LIN {X 0,Y 368.03,Z 575.323,A -85,B 0,C 180,E1 10655.932,E2 10655.932} C_VEL
LIN {X 0,Y 372.432,Z 552.778,A -85,B 0,C 180,E1 10654.833,E2 10654.833} C_VEL
LIN {X 0,Y 375.58,Z 532.541,A -85,B 0,C 180,E1 10654.081,E2 10654.081} C_VEL
LIN {X 0,Y 378.339,Z 507.8,A -85,B 0,C 180,E1 10653.405,E2 10653.405} C_VEL
LIN {X 0,Y 390.575,Z 315.874,A -85,B 0,C 180,E1 10649.482,E2 10649.482} C_VEL
LIN {X 0,Y 393.17,Z 275.11,A -85,B 0,C 180,E1 10648.652,E2 10648.652} C_VEL
LIN {X 0,Y 384.379,Z 261.212,A -85,B 0,C 180,E1 10645.871,E2 10645.871} C_VEL
LIN {X 0,Y 376.778,Z 250,A -85,B 0,C 180,E1 10643.167,E2 10643.167} C_VEL
LIN {X 0,Y 370.187,Z 240.873,A -85,B 0,C 180,E1 10640.515,E2 10640.515} C_VEL
LIN {X 0,Y 365.396,Z 234.593,A -85,B 0,C 180,E1 10638.341,E2 10638.341} C_VEL
LIN {X 0,Y 362.255,Z 230.576,A -85,B 0,C 180,E1 10636.764,E2 10636.764} C_VEL
LIN {X 0,Y 358.691,Z 226.093,A -85,B 0,C 180,E1 10634.777,E2 10634.777} C_VEL
LIN {X 0,Y 354.481,Z 220.931,A -85,B 0,C 180,E1 10632.047,E2 10632.047} C_VEL
LIN {X 0,Y 349.673,Z 215.334,A -85,B 0,C 180,E1 10628.054,E2 10628.054} C_VEL
LIN {X 0,Y 344.902,Z 210.541,A -85,B 0,C 180,E1 10620.996,E2 10620.996} C_VEL
LIN {X 0,Y 344.302,Z 209.98,A -85,B 0,C 180,E1 10617.836,E2 10617.836} C_VEL
LIN {X 0,Y 344.699,Z 211.471,A -85,B 0,C 180,E1 10614.006,E2 10614.006} C_VEL
LIN {X 0,Y 347.562,Z 215.069,A -85,B 0,C 180,E1 10608.799,E2 10608.799} C_VEL
LIN {X 0,Y 350.867,Z 219.711,A -85,B 0,C 180,E1 10605.308,E2 10605.308} C_VEL
LIN {X 0,Y 351.984,Z 221.296,A -85,B 0,C 180,E1 10604.344,E2 10604.344} C_VEL
LIN {X 0,Y 355.628,Z 226.333,A -85,B 0,C 180,E1 10601.645,E2 10601.645} C_VEL
LIN {X 0,Y 359.331,Z 231.448,A -85,B 0,C 180,E1 10599.348,E2 10599.348} C_VEL
LIN {X 0,Y 363.967,Z 237.983,A -85,B 0,C 180,E1 10596.869,E2 10596.869} C_VEL
LIN {X 0,Y 370.087,Z 246.981,A -85,B 0,C 180,E1 10594.044,E2 10594.044} C_VEL
LIN {X 0,Y 376.169,Z 256.349,A -85,B 0,C 180,E1 10591.589,E2 10591.589} C_VEL
LIN {X 0,Y 382.889,Z 267.209,A -85,B 0,C 180,E1 10589.171,E2 10589.171} C_VEL
LIN {X 0,Y 389.905,Z 279.202,A -85,B 0,C 180,E1 10586.892,E2 10586.892} C_VEL
LIN {X 0,Y 390.523,Z 280.623,A -85,B 0,C 180,E1 10586.69,E2 10586.69} C_VEL
LIN {X 0,Y 377.585,Z 508.657,A -85,B 0,C 180,E1 10582.319,E2 10582.319} C_VEL
LIN {X 0,Y 375.428,Z 530.973,A -85,B 0,C 180,E1 10581.772,E2 10581.772} C_VEL
LIN {X 0,Y 372.339,Z 551.704,A -85,B 0,C 180,E1 10581.048,E2 10581.048} C_VEL
LIN {X 0,Y 368.361,Z 572.767,A -85,B 0,C 180,E1 10580.066,E2 10580.066} C_VEL
LIN {X 0,Y 364.024,Z 591.67,A -85,B 0,C 180,E1 10578.945,E2 10578.945} C_VEL
LIN {X 0,Y 358.708,Z 611.311,A -85,B 0,C 180,E1 10577.497,E2 10577.497} C_VEL
LIN {X 0,Y 353.173,Z 629.571,A -85,B 0,C 180,E1 10575.857,E2 10575.857} C_VEL
LIN {X 0,Y 346.964,Z 647.622,A -85,B 0,C 180,E1 10573.871,E2 10573.871} C_VEL
LIN {X 0,Y 340.274,Z 665.618,A -85,B 0,C 180,E1 10571.471,E2 10571.471} C_VEL
LIN {X 0,Y 333.892,Z 681.773,A -85,B 0,C 180,E1 10568.868,E2 10568.868} C_VEL
LIN {X 0,Y 327.863,Z 696.153,A -85,B 0,C 180,E1 10566.055,E2 10566.055} C_VEL
LIN {X 0,Y 321.867,Z 710.299,A -85,B 0,C 180,E1 10562.718,E2 10562.718} C_VEL
LIN {X 0,Y 316.825,Z 722.338,A -85,B 0,C 180,E1 10559.284,E2 10559.284} C_VEL
LIN {X 0,Y 312.53,Z 732.875,A -85,B 0,C 180,E1 10555.587,E2 10555.587} C_VEL
LIN {X 0,Y 309.109,Z 742.014,A -85,B 0,C 180,E1 10551.638,E2 10551.638} C_VEL
LIN {X 0,Y 306.717,Z 749.426,A -85,B 0,C 180,E1 10547.647,E2 10547.647} C_VEL
LIN {X 0,Y 305.203,Z 755.071,A -85,B 0,C 180,E1 10543.643,E2 10543.643} C_VEL
LIN {X 0,Y 304.379,Z 759.395,A -85,B 0,C 180,E1 10539.453,E2 10539.453} C_VEL
LIN {X 0,Y 304.077,Z 761.943,A -85,B 0,C 180,E1 10535.661,E2 10535.661} C_VEL
LIN {X 0,Y 303.986,Z 763.224,A -85,B 0,C 180,E1 10531.696,E2 10531.696} C_VEL
LIN {X 0,Y 303.989,Z 763.215,A -85,B 0,C 180,E1 10528.115,E2 10528.115} C_VEL
LIN {X 0,Y 304.083,Z 761.893,A -85,B 0,C 180,E1 10524.15,E2 10524.15} C_VEL
LIN {X 0,Y 304.392,Z 759.324,A -85,B 0,C 180,E1 10520.356,E2 10520.356} C_VEL
LIN {X 0,Y 305.236,Z 754.954,A -85,B 0,C 180,E1 10516.165,E2 10516.165} C_VEL
LIN {X 0,Y 306.324,Z 750.737,A -85,B 0,C 180,E1 10513.119,E2 10513.119} C_VEL
LIN {X 0,Y 306.002,Z 748.668,A -85,B 0,C 180,E1 10511.721,E2 10511.721} C_VEL
LIN {X 0,Y 302.102,Z 742.719,A -85,B 0,C 180,E1 10507.942,E2 10507.942} C_VEL
LIN {X 0,Y 302.28,Z 740.45,A -85,B 0,C 180,E1 10506.752,E2 10506.752} C_VEL
LIN {X 0,Y 306.107,Z 730.963,A -85,B 0,C 180,E1 10502.788,E2 10502.788} C_VEL
LIN {X 0,Y 311.162,Z 719.337,A -85,B 0,C 180,E1 10498.847,E2 10498.847} C_VEL
LIN {X 0,Y 316.773,Z 706.845,A -85,B 0,C 180,E1 10495.38,E2 10495.38} C_VEL
LIN {X 0,Y 322.621,Z 693.621,A -85,B 0,C 180,E1 10492.373,E2 10492.373} C_VEL
LIN {X 0,Y 329.225,Z 678.283,A -85,B 0,C 180,E1 10489.466,E2 10489.466} C_VEL
LIN {X 0,Y 335.931,Z 662.054,A -85,B 0,C 180,E1 10486.917,E2 10486.917} C_VEL
LIN {X 0,Y 342.314,Z 645.186,A -85,B 0,C 180,E1 10484.744,E2 10484.744} C_VEL
LIN {X 0,Y 349.073,Z 625.729,A -85,B 0,C 180,E1 10482.674,E2 10482.674} C_VEL
LIN {X 0,Y 355.034,Z 606.549,A -85,B 0,C 180,E1 10481.01,E2 10481.01} C_VEL
LIN {X 0,Y 360.276,Z 586.779,A -85,B 0,C 180,E1 10479.636,E2 10479.636} C_VEL
LIN {X 0,Y 365.159,Z 564.965,A -85,B 0,C 180,E1 10478.43,E2 10478.43} C_VEL
LIN {X 0,Y 369.101,Z 543.179,A -85,B 0,C 180,E1 10477.517,E2 10477.517} C_VEL
LIN {X 0,Y 371.952,Z 521.251,A -85,B 0,C 180,E1 10476.867,E2 10476.867} C_VEL
LIN {X 0,Y 374.108,Z 491.918,A -85,B 0,C 180,E1 10476.246,E2 10476.246} C_VEL
LIN {X 0,Y 386.33,Z 284.515,A -85,B 0,C 180,E1 10472.262,E2 10472.262} C_VEL
LIN {X 0,Y 378.451,Z 270.786,A -85,B 0,C 180,E1 10469.564,E2 10469.564} C_VEL
LIN {X 0,Y 370.714,Z 258.332,A -85,B 0,C 180,E1 10466.555,E2 10466.555} C_VEL
LIN {X 0,Y 364.99,Z 249.636,A -85,B 0,C 180,E1 10464.004,E2 10464.004} C_VEL
LIN {X 0,Y 359.677,Z 241.804,A -85,B 0,C 180,E1 10461.271,E2 10461.271} C_VEL
LIN {X 0,Y 356.149,Z 236.756,A -85,B 0,C 180,E1 10459.176,E2 10459.176} C_VEL
LIN {X 0,Y 352.925,Z 232.202,A -85,B 0,C 180,E1 10456.966,E2 10456.966} C_VEL
LIN {X 0,Y 349.827,Z 227.657,A -85,B 0,C 180,E1 10454.398,E2 10454.398} C_VEL
LIN {X 0,Y 346.535,Z 223.028,A -85,B 0,C 180,E1 10450.81,E2 10450.81} C_VEL
LIN {X 0,Y 344.076,Z 219.991,A -85,B 0,C 180,E1 10446.34,E2 10446.34} C_VEL
LIN {X 0,Y 343.53,Z 218.311,A -85,B 0,C 180,E1 10442.336,E2 10442.336} C_VEL
LIN {X 0,Y 344.064,Z 218.755,A -85,B 0,C 180,E1 10439.168,E2 10439.168} C_VEL
LIN {X 0,Y 348.217,Z 222.986,A -85,B 0,C 180,E1 10432.576,E2 10432.576} C_VEL
LIN {X 0,Y 349.257,Z 224.156,A -85,B 0,C 180,E1 10431.522,E2 10431.522} C_VEL
LIN {X 0,Y 354.086,Z 229.86,A -85,B 0,C 180,E1 10427.608,E2 10427.608} C_VEL
LIN {X 0,Y 358.751,Z 235.756,A -85,B 0,C 180,E1 10424.647,E2 10424.647} C_VEL
LIN {X 0,Y 363.139,Z 241.45,A -85,B 0,C 180,E1 10422.287,E2 10422.287} C_VEL
LIN {X 0,Y 369.123,Z 249.401,A -85,B 0,C 180,E1 10419.507,E2 10419.507} C_VEL
LIN {X 0,Y 376.122,Z 259.55,A -85,B 0,C 180,E1 10416.666,E2 10416.666} C_VEL
LIN {X 0,Y 383.714,Z 271.114,A -85,B 0,C 180,E1 10413.956,E2 10413.956} C_VEL
LIN {X 0,Y 388.89,Z 279.747,A -85,B 0,C 180,E1 10412.261,E2 10412.261} C_VEL
LIN {X 0,Y 375.193,Z 488.195,A -85,B 0,C 180,E1 10408.022,E2 10408.022} C_VEL
LIN {X 0,Y 372.711,Z 518.69,A -85,B 0,C 180,E1 10407.334,E2 10407.334} C_VEL
LIN {X 0,Y 369.596,Z 541.745,A -85,B 0,C 180,E1 10406.622,E2 10406.622} C_VEL
LIN {X 0,Y 365.445,Z 564.474,A -85,B 0,C 180,E1 10405.646,E2 10405.646} C_VEL
LIN {X 0,Y 360.248,Z 587.797,A -85,B 0,C 180,E1 10404.349,E2 10404.349} C_VEL
LIN {X 0,Y 354.809,Z 608.696,A -85,B 0,C 180,E1 10402.89,E2 10402.89} C_VEL
LIN {X 0,Y 348.682,Z 629.121,A -85,B 0,C 180,E1 10401.125,E2 10401.125} C_VEL
LIN {X 0,Y 342.163,Z 648.952,A -85,B 0,C 180,E1 10399.057,E2 10399.057} C_VEL
LIN {X 0,Y 335.831,Z 666.622,A -85,B 0,C 180,E1 10396.837,E2 10396.837} C_VEL
LIN {X 0,Y 328.72,Z 685.312,A -85,B 0,C 180,E1 10394.027,E2 10394.027} C_VEL
LIN {X 0,Y 322.316,Z 701.724,A -85,B 0,C 180,E1 10391.079,E2 10391.079} C_VEL
LIN {X 0,Y 316.265,Z 716.75,A -85,B 0,C 180,E1 10387.829,E2 10387.829} C_VEL
LIN {X 0,Y 310.526,Z 731.331,A -85,B 0,C 180,E1 10384.073,E2 10384.073} C_VEL
LIN {X 0,Y 305.865,Z 743.789,A -85,B 0,C 180,E1 10380.225,E2 10380.225} C_VEL
LIN {X 0,Y 302.198,Z 754.312,A -85,B 0,C 180,E1 10376.282,E2 10376.282} C_VEL
LIN {X 0,Y 299.451,Z 763.498,A -85,B 0,C 180,E1 10372.166,E2 10372.166} C_VEL
LIN {X 0,Y 297.611,Z 770.879,A -85,B 0,C 180,E1 10368.004,E2 10368.004} C_VEL
LIN {X 0,Y 296.523,Z 776.987,A -85,B 0,C 180,E1 10363.652,E2 10363.652} C_VEL
LIN {X 0,Y 296.094,Z 780.812,A -85,B 0,C 180,E1 10359.917,E2 10359.917} C_VEL
LIN {X 0,Y 295.973,Z 783.478,A -85,B 0,C 180,E1 10356.206,E2 10356.206} C_VEL
LIN {X 0,Y 295.966,Z 784.977,A -85,B 0,C 180,E1 10352.13,E2 10352.13} C_VEL
LIN {X 0,Y 295.971,Z 785.074,A -85,B 0,C 180,E1 10348.645,E2 10348.645} C_VEL
LIN {X 0,Y 295.956,Z 784.128,A -85,B 0,C 180,E1 10345.155,E2 10345.155} C_VEL
LIN {X 0,Y 296.038,Z 781.654,A -85,B 0,C 180,E1 10341.062,E2 10341.062} C_VEL
LIN {X 0,Y 296.38,Z 778.076,A -85,B 0,C 180,E1 10337.334,E2 10337.334} C_VEL
LIN {X 0,Y 297.238,Z 772.774,A -85,B 0,C 180,E1 10333.185,E2 10333.185} C_VEL
LIN {X 0,Y 298.868,Z 765.608,A -85,B 0,C 180,E1 10328.969,E2 10328.969} C_VEL
LIN {X 0,Y 301.477,Z 756.611,A -85,B 0,C 180,E1 10324.671,E2 10324.671} C_VEL
LIN {X 0,Y 304.866,Z 746.485,A -85,B 0,C 180,E1 10320.737,E2 10320.737} C_VEL
LIN {X 0,Y 309.498,Z 733.937,A -85,B 0,C 180,E1 10316.689,E2 10316.689} C_VEL
LIN {X 0,Y 314.73,Z 720.655,A -85,B 0,C 180,E1 10313.101,E2 10313.101} C_VEL
LIN {X 0,Y 320.576,Z 705.886,A -85,B 0,C 180,E1 10309.789,E2 10309.789} C_VEL
LIN {X 0,Y 327.099,Z 689.449,A -85,B 0,C 180,E1 10306.677,E2 10306.677} C_VEL
LIN {X 0,Y 333.306,Z 673.234,A -85,B 0,C 180,E1 10304.103,E2 10304.103} C_VEL
LIN {X 0,Y 340.192,Z 654.371,A -85,B 0,C 180,E1 10301.597,E2 10301.597} C_VEL
LIN {X 0,Y 346.634,Z 635.528,A -85,B 0,C 180,E1 10299.504,E2 10299.504} C_VEL
LIN {X 0,Y 352.633,Z 615.965,A -85,B 0,C 180,E1 10297.716,E2 10297.716} C_VEL
LIN {X 0,Y 358.134,Z 596.262,A -85,B 0,C 180,E1 10296.213,E2 10296.213} C_VEL
LIN {X 0,Y 363.003,Z 575.753,A -85,B 0,C 180,E1 10294.954,E2 10294.954} C_VEL
LIN {X 0,Y 367.47,Z 553.785,A -85,B 0,C 180,E1 10293.874,E2 10293.874} C_VEL
LIN {X 0,Y 370.785,Z 533.196,A -85,B 0,C 180,E1 10293.103,E2 10293.103} C_VEL
LIN {X 0,Y 373.66,Z 508.504,A -85,B 0,C 180,E1 10292.422,E2 10292.422} C_VEL
LIN {X 0,Y 386.203,Z 318.554,A -85,B 0,C 180,E1 10288.527,E2 10288.527} C_VEL
LIN {X 0,Y 388.714,Z 279.297,A -85,B 0,C 180,E1 10287.705,E2 10287.705} C_VEL
LIN {X 0,Y 380.162,Z 265.668,A -85,B 0,C 180,E1 10284.858,E2 10284.858} C_VEL
LIN {X 0,Y 371.938,Z 253.409,A -85,B 0,C 180,E1 10281.734,E2 10281.734} C_VEL
LIN {X 0,Y 364.697,Z 243.494,A -85,B 0,C 180,E1 10278.543,E2 10278.543} C_VEL
LIN {X 0,Y 360.39,Z 237.928,A -85,B 0,C 180,E1 10276.355,E2 10276.355} C_VEL
LIN {X 0,Y 357.044,Z 233.634,A -85,B 0,C 180,E1 10274.432,E2 10274.432} C_VEL
LIN {X 0,Y 353.047,Z 228.624,A -85,B 0,C 180,E1 10271.765,E2 10271.765} C_VEL
LIN {X 0,Y 348.527,Z 223.207,A -85,B 0,C 180,E1 10267.915,E2 10267.915} C_VEL
LIN {X 0,Y 343.873,Z 218.424,A -85,B 0,C 180,E1 10260.833,E2 10260.833} C_VEL
LIN {X 0,Y 343.32,Z 217.931,A -85,B 0,C 180,E1 10257.663,E2 10257.663} C_VEL
LIN {X 0,Y 343.825,Z 219.685,A -85,B 0,C 180,E1 10253.655,E2 10253.655} C_VEL
LIN {X 0,Y 346.399,Z 222.9,A -85,B 0,C 180,E1 10249.017,E2 10249.017} C_VEL
LIN {X 0,Y 349.73,Z 227.605,A -85,B 0,C 180,E1 10245.428,E2 10245.428} C_VEL
LIN {X 0,Y 354.082,Z 233.9,A -85,B 0,C 180,E1 10241.988,E2 10241.988} C_VEL
LIN {X 0,Y 357.7,Z 239.039,A -85,B 0,C 180,E1 10239.677,E2 10239.677} C_VEL
LIN {X 0,Y 362.132,Z 245.409,A -85,B 0,C 180,E1 10237.244,E2 10237.244} C_VEL
LIN {X 0,Y 368.105,Z 254.397,A -85,B 0,C 180,E1 10234.413,E2 10234.413} C_VEL
LIN {X 0,Y 374.923,Z 265.093,A -85,B 0,C 180,E1 10231.617,E2 10231.617} C_VEL
LIN {X 0,Y 382.618,Z 278.019,A -85,B 0,C 180,E1 10228.841,E2 10228.841} C_VEL
LIN {X 0,Y 386.222,Z 284.81,A -85,B 0,C 180,E1 10227.633,E2 10227.633} C_VEL
LIN {X 0,Y 372.875,Z 510.263,A -85,B 0,C 180,E1 10223.289,E2 10223.289} C_VEL
LIN {X 0,Y 370.464,Z 533.064,A -85,B 0,C 180,E1 10222.709,E2 10222.709} C_VEL
LIN {X 0,Y 367.326,Z 553.251,A -85,B 0,C 180,E1 10221.99,E2 10221.99} C_VEL
LIN {X 0,Y 363.3,Z 573.556,A -85,B 0,C 180,E1 10221.029,E2 10221.029} C_VEL
LIN {X 0,Y 358.531,Z 593.601,A -85,B 0,C 180,E1 10219.827,E2 10219.827} C_VEL
LIN {X 0,Y 352.879,Z 613.422,A -85,B 0,C 180,E1 10218.328,E2 10218.328} C_VEL
LIN {X 0,Y 346.543,Z 633.073,A -85,B 0,C 180,E1 10216.496,E2 10216.496} C_VEL
LIN {X 0,Y 340.245,Z 650.696,A -85,B 0,C 180,E1 10214.495,E2 10214.495} C_VEL
LIN {X 0,Y 333.634,Z 667.524,A -85,B 0,C 180,E1 10212.166,E2 10212.166} C_VEL
LIN {X 0,Y 326.963,Z 683.557,A -85,B 0,C 180,E1 10209.498,E2 10209.498} C_VEL
LIN {X 0,Y 320.947,Z 697.338,A -85,B 0,C 180,E1 10206.736,E2 10206.736} C_VEL
LIN {X 0,Y 315.012,Z 710.641,A -85,B 0,C 180,E1 10203.523,E2 10203.523} C_VEL
LIN {X 0,Y 309.701,Z 722.665,A -85,B 0,C 180,E1 10200.026,E2 10200.026} C_VEL
LIN {X 0,Y 305.16,Z 733.199,A -85,B 0,C 180,E1 10196.252,E2 10196.252} C_VEL
LIN {X 0,Y 301.52,Z 742.327,A -85,B 0,C 180,E1 10192.211,E2 10192.211} C_VEL
LIN {X 0,Y 298.956,Z 749.731,A -85,B 0,C 180,E1 10188.121,E2 10188.121} C_VEL
LIN {X 0,Y 297.323,Z 755.373,A -85,B 0,C 180,E1 10184.012,E2 10184.012} C_VEL
LIN {X 0,Y 296.427,Z 759.691,A -85,B 0,C 180,E1 10179.709,E2 10179.709} C_VEL
LIN {X 0,Y 296.093,Z 762.237,A -85,B 0,C 180,E1 10175.814,E2 10175.814} C_VEL
LIN {X 0,Y 295.992,Z 763.515,A -85,B 0,C 180,E1 10171.742,E2 10171.742} C_VEL
LIN {X 0,Y 295.994,Z 763.526,A -85,B 0,C 180,E1 10168.258,E2 10168.258} C_VEL
LIN {X 0,Y 296.089,Z 762.292,A -85,B 0,C 180,E1 10164.186,E2 10164.186} C_VEL
LIN {X 0,Y 296.412,Z 759.769,A -85,B 0,C 180,E1 10160.29,E2 10160.29} C_VEL
LIN {X 0,Y 297.359,Z 755.254,A -85,B 0,C 180,E1 10155.791,E2 10155.791} C_VEL
LIN {X 0,Y 299.015,Z 749.588,A -85,B 0,C 180,E1 10151.681,E2 10151.681} C_VEL
LIN {X 0,Y 301.605,Z 742.133,A -85,B 0,C 180,E1 10147.59,E2 10147.59} C_VEL
LIN {X 0,Y 302.28,Z 740.45,A -85,B 0,C 180,E1 10146.752,E2 10146.752} C_VEL
LIN {X 0,Y 302.486,Z 737.71,A -85,B 0,C 180,E1 10145.376,E2 10145.376} C_VEL
LIN {X 0,Y 300.12,Z 730.017,A -85,B 0,C 180,E1 10141.634,E2 10141.634} C_VEL
LIN {X 0,Y 300.759,Z 727.058,A -85,B 0,C 180,E1 10140.501,E2 10140.501} C_VEL
LIN {X 0,Y 306.243,Z 715.364,A -85,B 0,C 180,E1 10136.736,E2 10136.736} C_VEL
LIN {X 0,Y 312.14,Z 702.702,A -85,B 0,C 180,E1 10133.431,E2 10133.431} C_VEL
LIN {X 0,Y 319.23,Z 687.304,A -85,B 0,C 180,E1 10130.118,E2 10130.118} C_VEL
LIN {X 0,Y 326.173,Z 671.688,A -85,B 0,C 180,E1 10127.356,E2 10127.356} C_VEL
LIN {X 0,Y 332.899,Z 655.333,A -85,B 0,C 180,E1 10124.984,E2 10124.984} C_VEL
LIN {X 0,Y 339.889,Z 636.967,A -85,B 0,C 180,E1 10122.783,E2 10122.783} C_VEL
LIN {X 0,Y 346.384,Z 618.198,A -85,B 0,C 180,E1 10120.939,E2 10120.939} C_VEL
LIN {X 0,Y 352.092,Z 599.148,A -85,B 0,C 180,E1 10119.431,E2 10119.431} C_VEL
LIN {X 0,Y 357.576,Z 578.029,A -85,B 0,C 180,E1 10118.084,E2 10118.084} C_VEL
LIN {X 0,Y 361.727,Z 558.766,A -85,B 0,C 180,E1 10117.115,E2 10117.115} C_VEL
LIN {X 0,Y 365.378,Z 537.264,A -85,B 0,C 180,E1 10116.297,E2 10116.297} C_VEL
LIN {X 0,Y 368.092,Z 515.346,A -85,B 0,C 180,E1 10115.693,E2 10115.693} C_VEL
LIN {X 0,Y 375.18,Z 399.549,A -85,B 0,C 180,E1 10113.432,E2 10113.432} C_VEL
LIN {X 0,Y 382.145,Z 288.685,A -85,B 0,C 180,E1 10111.298,E2 10111.298} C_VEL
LIN {X 0,Y 374.329,Z 275.003,A -85,B 0,C 180,E1 10108.476,E2 10108.476} C_VEL
LIN {X 0,Y 366.684,Z 262.542,A -85,B 0,C 180,E1 10105.304,E2 10105.304} C_VEL
LIN {X 0,Y 360.625,Z 253.213,A -85,B 0,C 180,E1 10102.367,E2 10102.367} C_VEL
LIN {X 0,Y 357.213,Z 248.275,A -85,B 0,C 180,E1 10100.48,E2 10100.48} C_VEL
LIN {X 0,Y 354.454,Z 244.161,A -85,B 0,C 180,E1 10098.758,E2 10098.758} C_VEL
LIN {X 0,Y 351.322,Z 239.643,A -85,B 0,C 180,E1 10096.535,E2 10096.535} C_VEL
LIN {X 0,Y 348.335,Z 235.208,A -85,B 0,C 180,E1 10093.952,E2 10093.952} C_VEL
LIN {X 0,Y 345.275,Z 230.594,A -85,B 0,C 180,E1 10090.428,E2 10090.428} C_VEL
LIN {X 0,Y 342.577,Z 226.627,A -85,B 0,C 180,E1 10083.682,E2 10083.682} C_VEL
LIN {X 0,Y 342.76,Z 226.314,A -85,B 0,C 180,E1 10080.502,E2 10080.502} C_VEL
LIN {X 0,Y 344.521,Z 228.504,A -85,B 0,C 180,E1 10076.006,E2 10076.006} C_VEL
LIN {X 0,Y 347.865,Z 231.702,A -85,B 0,C 180,E1 10071.904,E2 10071.904} C_VEL
LIN {X 0,Y 352.641,Z 237.555,A -85,B 0,C 180,E1 10067.889,E2 10067.889} C_VEL
LIN {X 0,Y 357.085,Z 243.288,A -85,B 0,C 180,E1 10064.989,E2 10064.989} C_VEL
LIN {X 0,Y 361.383,Z 248.999,A -85,B 0,C 180,E1 10062.614,E2 10062.614} C_VEL
LIN {X 0,Y 367.013,Z 256.652,A -85,B 0,C 180,E1 10059.924,E2 10059.924} C_VEL
LIN {X 0,Y 373.867,Z 266.827,A -85,B 0,C 180,E1 10057.059,E2 10057.059} C_VEL
LIN {X 0,Y 381.029,Z 277.988,A -85,B 0,C 180,E1 10054.427,E2 10054.427} C_VEL
LIN {X 0,Y 384.609,Z 284.061,A -85,B 0,C 180,E1 10053.207,E2 10053.207} C_VEL
LIN {X 0,Y 370.454,Z 492.545,A -85,B 0,C 180,E1 10048.958,E2 10048.958} C_VEL
LIN {X 0,Y 368.064,Z 519.686,A -85,B 0,C 180,E1 10048.331,E2 10048.331} C_VEL
LIN {X 0,Y 364.839,Z 542.581,A -85,B 0,C 180,E1 10047.618,E2 10047.618} C_VEL
LIN {X 0,Y 360.591,Z 565.067,A -85,B 0,C 180,E1 10046.646,E2 10046.646} C_VEL
LIN {X 0,Y 355.227,Z 588.262,A -85,B 0,C 180,E1 10045.35,E2 10045.35} C_VEL
LIN {X 0,Y 349.525,Z 609.415,A -85,B 0,C 180,E1 10043.865,E2 10043.865} C_VEL
LIN {X 0,Y 343.279,Z 629.417,A -85,B 0,C 180,E1 10042.121,E2 10042.121} C_VEL
LIN {X 0,Y 336.52,Z 649.173,A -85,B 0,C 180,E1 10040.044,E2 10040.044} C_VEL
LIN {X 0,Y 330.017,Z 666.624,A -85,B 0,C 180,E1 10037.832,E2 10037.832} C_VEL
LIN {X 0,Y 322.785,Z 684.85,A -85,B 0,C 180,E1 10035.07,E2 10035.07} C_VEL
LIN {X 0,Y 316.095,Z 701.184,A -85,B 0,C 180,E1 10032.111,E2 10032.111} C_VEL
LIN {X 0,Y 309.671,Z 716.386,A -85,B 0,C 180,E1 10028.782,E2 10028.782} C_VEL
LIN {X 0,Y 303.597,Z 730.986,A -85,B 0,C 180,E1 10024.962,E2 10024.962} C_VEL
LIN {X 0,Y 298.86,Z 742.852,A -85,B 0,C 180,E1 10021.235,E2 10021.235} C_VEL
LIN {X 0,Y 294.759,Z 753.905,A -85,B 0,C 180,E1 10017.035,E2 10017.035} C_VEL
LIN {X 0,Y 291.776,Z 763.182,A -85,B 0,C 180,E1 10012.781,E2 10012.781} C_VEL
LIN {X 0,Y 289.773,Z 770.568,A -85,B 0,C 180,E1 10008.508,E2 10008.508} C_VEL
LIN {X 0,Y 288.586,Z 776.685,A -85,B 0,C 180,E1 10004.035,E2 10004.035} C_VEL
LIN {X 0,Y 288.112,Z 780.514,A -85,B 0,C 180,E1 10000.194,E2 10000.194} C_VEL
LIN {X 0,Y 287.98,Z 783.184,A -85,B 0,C 180,E1 9996.379,E2 9996.379} C_VEL
LIN {X 0,Y 287.972,Z 784.686,A -85,B 0,C 180,E1 9992.189,E2 9992.189} C_VEL
LIN {X 0,Y 287.976,Z 784.783,A -85,B 0,C 180,E1 9988.607,E2 9988.607} C_VEL
LIN {X 0,Y 287.96,Z 783.835,A -85,B 0,C 180,E1 9985.02,E2 9985.02} C_VEL
LIN {X 0,Y 288.052,Z 781.355,A -85,B 0,C 180,E1 9980.812,E2 9980.812} C_VEL
LIN {X 0,Y 288.433,Z 777.719,A -85,B 0,C 180,E1 9976.928,E2 9976.928} C_VEL
LIN {X 0,Y 289.435,Z 772.15,A -85,B 0,C 180,E1 9972.51,E2 9972.51} C_VEL
LIN {X 0,Y 291.204,Z 765.021,A -85,B 0,C 180,E1 9968.234,E2 9968.234} C_VEL
LIN {X 0,Y 294.101,Z 755.802,A -85,B 0,C 180,E1 9963.772,E2 9963.772} C_VEL
LIN {X 0,Y 297.565,Z 746.177,A -85,B 0,C 180,E1 9959.957,E2 9959.957} C_VEL
LIN {X 0,Y 302.512,Z 733.586,A -85,B 0,C 180,E1 9955.815,E2 9955.815} C_VEL
LIN {X 0,Y 308.046,Z 720.296,A -85,B 0,C 180,E1 9952.161,E2 9952.161} C_VEL
LIN {X 0,Y 314.21,Z 705.506,A -85,B 0,C 180,E1 9948.801,E2 9948.801} C_VEL
LIN {X 0,Y 321.15,Z 688.781,A -85,B 0,C 180,E1 9945.606,E2 9945.606} C_VEL
LIN {X 0,Y 327.837,Z 672.109,A -85,B 0,C 180,E1 9942.95,E2 9942.95} C_VEL
LIN {X 0,Y 334.705,Z 653.97,A -85,B 0,C 180,E1 9940.541,E2 9940.541} C_VEL
LIN {X 0,Y 341.426,Z 635.027,A -85,B 0,C 180,E1 9938.432,E2 9938.432} C_VEL
LIN {X 0,Y 347.646,Z 615.379,A -85,B 0,C 180,E1 9936.64,E2 9936.64} C_VEL
LIN {X 0,Y 353.615,Z 594.404,A -85,B 0,C 180,E1 9935.06,E2 9935.06} C_VEL
LIN {X 0,Y 358.325,Z 575.148,A -85,B 0,C 180,E1 9933.89,E2 9933.89} C_VEL
LIN {X 0,Y 363.015,Z 552.479,A -85,B 0,C 180,E1 9932.792,E2 9932.792} C_VEL
LIN {X 0,Y 366.36,Z 532.171,A -85,B 0,C 180,E1 9932.044,E2 9932.044} C_VEL
LIN {X 0,Y 369.227,Z 507.637,A -85,B 0,C 180,E1 9931.378,E2 9931.378} C_VEL
LIN {X 0,Y 382.384,Z 314.913,A -85,B 0,C 180,E1 9927.422,E2 9927.422} C_VEL
LIN {X 0,Y 384.442,Z 283.695,A -85,B 0,C 180,E1 9926.765,E2 9926.765} C_VEL
LIN {X 0,Y 376.655,Z 271.153,A -85,B 0,C 180,E1 9924.046,E2 9924.046} C_VEL
LIN {X 0,Y 369.412,Z 260.193,A -85,B 0,C 180,E1 9921.182,E2 9921.182} C_VEL
LIN {X 0,Y 362.752,Z 250.837,A -85,B 0,C 180,E1 9918.147,E2 9918.147} C_VEL
LIN {X 0,Y 358.269,Z 244.929,A -85,B 0,C 180,E1 9915.789,E2 9915.789} C_VEL
LIN {X 0,Y 355.283,Z 241.035,A -85,B 0,C 180,E1 9914.006,E2 9914.006} C_VEL
LIN {X 0,Y 351.619,Z 236.315,A -85,B 0,C 180,E1 9911.481,E2 9911.481} C_VEL
LIN {X 0,Y 347.219,Z 230.963,A -85,B 0,C 180,E1 9907.612,E2 9907.612} C_VEL
LIN {X 0,Y 342.846,Z 226.309,A -85,B 0,C 180,E1 9900.668,E2 9900.668} C_VEL
LIN {X 0,Y 342.346,Z 225.875,A -85,B 0,C 180,E1 9897.656,E2 9897.656} C_VEL
LIN {X 0,Y 342.854,Z 227.682,A -85,B 0,C 180,E1 9893.637,E2 9893.637} C_VEL
LIN {X 0,Y 345.243,Z 230.735,A -85,B 0,C 180,E1 9889.234,E2 9889.234} C_VEL
LIN {X 0,Y 349.024,Z 236.245,A -85,B 0,C 180,E1 9885.144,E2 9885.144} C_VEL
LIN {X 0,Y 352.658,Z 241.65,A -85,B 0,C 180,E1 9882.255,E2 9882.255} C_VEL
LIN {X 0,Y 356.086,Z 246.628,A -85,B 0,C 180,E1 9880.009,E2 9880.009} C_VEL
LIN {X 0,Y 360.404,Z 252.968,A -85,B 0,C 180,E1 9877.575,E2 9877.575} C_VEL
LIN {X 0,Y 366.471,Z 262.304,A -85,B 0,C 180,E1 9874.637,E2 9874.637} C_VEL
LIN {X 0,Y 373.845,Z 274.313,A -85,B 0,C 180,E1 9871.571,E2 9871.571} C_VEL
LIN {X 0,Y 381.204,Z 287.19,A -85,B 0,C 180,E1 9868.888,E2 9868.888} C_VEL
LIN {X 0,Y 382.029,Z 288.917,A -85,B 0,C 180,E1 9868.597,E2 9868.597} C_VEL
LIN {X 0,Y 368.298,Z 511.552,A -85,B 0,C 180,E1 9864.29,E2 9864.29} C_VEL
LIN {X 0,Y 365.603,Z 535.15,A -85,B 0,C 180,E1 9863.672,E2 9863.672} C_VEL
LIN {X 0,Y 362.223,Z 555.934,A -85,B 0,C 180,E1 9862.912,E2 9862.912} C_VEL
LIN {X 0,Y 357.89,Z 576.317,A -85,B 0,C 180,E1 9861.911,E2 9861.911} C_VEL
LIN {X 0,Y 352.563,Z 597.265,A -85,B 0,C 180,E1 9860.604,E2 9860.604} C_VEL
LIN {X 0,Y 346.986,Z 615.99,A -85,B 0,C 180,E1 9859.147,E2 9859.147} C_VEL
LIN {X 0,Y 340.58,Z 634.856,A -85,B 0,C 180,E1 9857.34,E2 9857.34} C_VEL
LIN {X 0,Y 333.993,Z 652.511,A -85,B 0,C 180,E1 9855.291,E2 9855.291} C_VEL
LIN {X 0,Y 327.214,Z 669.013,A -85,B 0,C 180,E1 9852.953,E2 9852.953} C_VEL
LIN {X 0,Y 320.308,Z 684.83,A -85,B 0,C 180,E1 9850.251,E2 9850.251} C_VEL
LIN {X 0,Y 313.715,Z 699.339,A -85,B 0,C 180,E1 9847.268,E2 9847.268} C_VEL
LIN {X 0,Y 307.588,Z 712.339,A -85,B 0,C 180,E1 9843.993,E2 9843.993} C_VEL
LIN {X 0,Y 301.68,Z 724.991,A -85,B 0,C 180,E1 9840.113,E2 9840.113} C_VEL
LIN {X 0,Y 297.217,Z 734.999,A -85,B 0,C 180,E1 9836.362,E2 9836.362} C_VEL
LIN {X 0,Y 293.503,Z 743.801,A -85,B 0,C 180,E1 9832.218,E2 9832.218} C_VEL
LIN {X 0,Y 290.757,Z 751.328,A -85,B 0,C 180,E1 9827.72,E2 9827.72} C_VEL
LIN {X 0,Y 289.165,Z 756.856,A -85,B 0,C 180,E1 9823.395,E2 9823.395} C_VEL
LIN {X 0,Y 288.369,Z 760.588,A -85,B 0,C 180,E1 9819.177,E2 9819.177} C_VEL
LIN {X 0,Y 288.066,Z 762.975,A -85,B 0,C 180,E1 9814.978,E2 9814.978} C_VEL
LIN {X 0,Y 287.998,Z 763.869,A -85,B 0,C 180,E1 9811.194,E2 9811.194} C_VEL
LIN {X 0,Y 288.012,Z 763.706,A -85,B 0,C 180,E1 9807.214,E2 9807.214} C_VEL
LIN {X 0,Y 288.15,Z 762.157,A -85,B 0,C 180,E1 9803.225,E2 9803.225} C_VEL
LIN {X 0,Y 288.618,Z 759.296,A -85,B 0,C 180,E1 9799.016,E2 9799.016} C_VEL
LIN {X 0,Y 289.69,Z 754.83,A -85,B 0,C 180,E1 9794.793,E2 9794.793} C_VEL
LIN {X 0,Y 291.838,Z 748.225,A -85,B 0,C 180,E1 9790.174,E2 9790.174} C_VEL
LIN {X 0,Y 294.887,Z 740.496,A -85,B 0,C 180,E1 9785.992,E2 9785.992} C_VEL
LIN {X 0,Y 299.067,Z 730.785,A -85,B 0,C 180,E1 9781.876,E2 9781.876} C_VEL
LIN {X 0,Y 300.759,Z 727.058,A -85,B 0,C 180,E1 9780.501,E2 9780.501} C_VEL
LIN {X 0,Y 301.504,Z 723.613,A -85,B 0,C 180,E1 9779.191,E2 9779.191} C_VEL
LIN {X 0,Y 300.721,Z 714.288,A -85,B 0,C 180,E1 9775.563,E2 9775.563} C_VEL
LIN {X 0,Y 301.815,Z 710.761,A -85,B 0,C 180,E1 9774.5,E2 9774.5} C_VEL
LIN {X 0,Y 308.848,Z 696.414,A -85,B 0,C 180,E1 9770.985,E2 9770.985} C_VEL
LIN {X 0,Y 315.943,Z 681.516,A -85,B 0,C 180,E1 9767.986,E2 9767.986} C_VEL
LIN {X 0,Y 323.062,Z 665.568,A -85,B 0,C 180,E1 9765.369,E2 9765.369} C_VEL
LIN {X 0,Y 330.538,Z 647.606,A -85,B 0,C 180,E1 9762.944,E2 9762.944} C_VEL
LIN {X 0,Y 337.467,Z 629.44,A -85,B 0,C 180,E1 9760.931,E2 9760.931} C_VEL
LIN {X 0,Y 343.602,Z 611.126,A -85,B 0,C 180,E1 9759.284,E2 9759.284} C_VEL
LIN {X 0,Y 349.719,Z 590.368,A -85,B 0,C 180,E1 9757.768,E2 9757.768} C_VEL
LIN {X 0,Y 354.83,Z 569.858,A -85,B 0,C 180,E1 9756.576,E2 9756.576} C_VEL
LIN {X 0,Y 359.098,Z 548.32,A -85,B 0,C 180,E1 9755.626,E2 9755.626} C_VEL
LIN {X 0,Y 362.622,Z 524.952,A -85,B 0,C 180,E1 9754.879,E2 9754.879} C_VEL
LIN {X 0,Y 364.754,Z 502.277,A -85,B 0,C 180,E1 9754.361,E2 9754.361} C_VEL
LIN {X 0,Y 378.032,Z 292.993,A -85,B 0,C 180,E1 9750.31,E2 9750.31} C_VEL
LIN {X 0,Y 370.777,Z 280.1,A -85,B 0,C 180,E1 9747.547,E2 9747.547} C_VEL
LIN {X 0,Y 364.153,Z 269.09,A -85,B 0,C 180,E1 9744.668,E2 9744.668} C_VEL
LIN {X 0,Y 358.282,Z 259.822,A -85,B 0,C 180,E1 9741.693,E2 9741.693} C_VEL
LIN {X 0,Y 353.255,Z 252.174,A -85,B 0,C 180,E1 9738.653,E2 9738.653} C_VEL
LIN {X 0,Y 349.743,Z 247.08,A -85,B 0,C 180,E1 9736.1,E2 9736.1} C_VEL
LIN {X 0,Y 347.032,Z 242.927,A -85,B 0,C 180,E1 9733.666,E2 9733.666} C_VEL
LIN {X 0,Y 343.792,Z 238.012,A -85,B 0,C 180,E1 9729.711,E2 9729.711} C_VEL
LIN {X 0,Y 341.581,Z 234.478,A -85,B 0,C 180,E1 9723.356,E2 9723.356} C_VEL
LIN {X 0,Y 341.849,Z 234.35,A -85,B 0,C 180,E1 9720.168,E2 9720.168} C_VEL
LIN {X 0,Y 344.082,Z 237.028,A -85,B 0,C 180,E1 9715.166,E2 9715.166} C_VEL
LIN {X 0,Y 346.637,Z 239.509,A -85,B 0,C 180,E1 9712.125,E2 9712.125} C_VEL
LIN {X 0,Y 351.206,Z 245.249,A -85,B 0,C 180,E1 9708.172,E2 9708.172} C_VEL
LIN {X 0,Y 355.557,Z 251.002,A -85,B 0,C 180,E1 9705.257,E2 9705.257} C_VEL
LIN {X 0,Y 359.93,Z 256.938,A -85,B 0,C 180,E1 9702.792,E2 9702.792} C_VEL
LIN {X 0,Y 365.555,Z 264.917,A -85,B 0,C 180,E1 9700.049,E2 9700.049} C_VEL
LIN {X 0,Y 371.81,Z 274.379,A -85,B 0,C 180,E1 9697.384,E2 9697.384} C_VEL
LIN {X 0,Y 378.564,Z 285.195,A -85,B 0,C 180,E1 9694.835,E2 9694.835} C_VEL
LIN {X 0,Y 380.424,Z 288.572,A -85,B 0,C 180,E1 9694.17,E2 9694.17} C_VEL
LIN {X 0,Y 365.857,Z 496.298,A -85,B 0,C 180,E1 9689.93,E2 9689.93} C_VEL
LIN {X 0,Y 363.531,Z 520.693,A -85,B 0,C 180,E1 9689.354,E2 9689.354} C_VEL
LIN {X 0,Y 360.133,Z 543.707,A -85,B 0,C 180,E1 9688.627,E2 9688.627} C_VEL
LIN {X 0,Y 356.006,Z 564.921,A -85,B 0,C 180,E1 9687.709,E2 9687.709} C_VEL
LIN {X 0,Y 350.461,Z 588.196,A -85,B 0,C 180,E1 9686.413,E2 9686.413} C_VEL
LIN {X 0,Y 344.537,Z 609.468,A -85,B 0,C 180,E1 9684.92,E2 9684.92} C_VEL
LIN {X 0,Y 338.098,Z 629.374,A -85,B 0,C 180,E1 9683.182,E2 9683.182} C_VEL
LIN {X 0,Y 331.03,Z 649.273,A -85,B 0,C 180,E1 9681.079,E2 9681.079} C_VEL
LIN {X 0,Y 324.165,Z 666.993,A -85,B 0,C 180,E1 9678.814,E2 9678.814} C_VEL
LIN {X 0,Y 316.685,Z 685.036,A -85,B 0,C 180,E1 9676.041,E2 9676.041} C_VEL
LIN {X 0,Y 309.92,Z 700.799,A -85,B 0,C 180,E1 9673.152,E2 9673.152} C_VEL
LIN {X 0,Y 303.163,Z 716.025,A -85,B 0,C 180,E1 9669.778,E2 9669.778} C_VEL
LIN {X 0,Y 297.038,Z 729.984,A -85,B 0,C 180,E1 9666.09,E2 9666.09} C_VEL
LIN {X 0,Y 291.953,Z 741.919,A -85,B 0,C 180,E1 9662.292,E2 9662.292} C_VEL
LIN {X 0,Y 287.461,Z 753.246,A -85,B 0,C 180,E1 9657.937,E2 9657.937} C_VEL
LIN {X 0,Y 284.254,Z 762.464,A -85,B 0,C 180,E1 9653.64,E2 9653.64} C_VEL
LIN {X 0,Y 282.04,Z 769.939,A -85,B 0,C 180,E1 9649.25,E2 9649.25} C_VEL
LIN {X 0,Y 280.745,Z 775.934,A -85,B 0,C 180,E1 9644.858,E2 9644.858} C_VEL
LIN {X 0,Y 280.136,Z 780.217,A -85,B 0,C 180,E1 9640.488,E2 9640.488} C_VEL
LIN {X 0,Y 279.988,Z 782.89,A -85,B 0,C 180,E1 9636.562,E2 9636.562} C_VEL
LIN {X 0,Y 279.976,Z 784.395,A -85,B 0,C 180,E1 9632.251,E2 9632.251} C_VEL
LIN {X 0,Y 279.98,Z 784.492,A -85,B 0,C 180,E1 9628.568,E2 9628.568} C_VEL
LIN {X 0,Y 279.963,Z 783.543,A -85,B 0,C 180,E1 9624.878,E2 9624.878} C_VEL
LIN {X 0,Y 280.068,Z 781.057,A -85,B 0,C 180,E1 9620.548,E2 9620.548} C_VEL
LIN {X 0,Y 280.477,Z 777.471,A -85,B 0,C 180,E1 9616.602,E2 9616.602} C_VEL
LIN {X 0,Y 281.546,Z 772.025,A -85,B 0,C 180,E1 9612.128,E2 9612.128} C_VEL
LIN {X 0,Y 283.391,Z 765.075,A -85,B 0,C 180,E1 9607.821,E2 9607.821} C_VEL
LIN {X 0,Y 286.365,Z 756.226,A -85,B 0,C 180,E1 9603.359,E2 9603.359} C_VEL
LIN {X 0,Y 290.113,Z 746.38,A -85,B 0,C 180,E1 9599.332,E2 9599.332} C_VEL
LIN {X 0,Y 295.502,Z 733.462,A -85,B 0,C 180,E1 9594.967,E2 9594.967} C_VEL
LIN {X 0,Y 301.452,Z 719.939,A -85,B 0,C 180,E1 9591.181,E2 9591.181} C_VEL
LIN {X 0,Y 307.995,Z 705.008,A -85,B 0,C 180,E1 9587.745,E2 9587.745} C_VEL
LIN {X 0,Y 315.364,Z 688.03,A -85,B 0,C 180,E1 9584.481,E2 9584.481} C_VEL
LIN {X 0,Y 322.307,Z 671.477,A -85,B 0,C 180,E1 9581.833,E2 9581.833} C_VEL
LIN {X 0,Y 329.416,Z 653.363,A -85,B 0,C 180,E1 9579.426,E2 9579.426} C_VEL
LIN {X 0,Y 336.305,Z 634.614,A -85,B 0,C 180,E1 9577.337,E2 9577.337} C_VEL
LIN {X 0,Y 342.784,Z 614.8,A -85,B 0,C 180,E1 9575.533,E2 9575.533} C_VEL
LIN {X 0,Y 349.049,Z 593.317,A -85,B 0,C 180,E1 9573.929,E2 9573.929} C_VEL
LIN {X 0,Y 354.13,Z 573.053,A -85,B 0,C 180,E1 9572.716,E2 9572.716} C_VEL
LIN {X 0,Y 358.921,Z 549.884,A -85,B 0,C 180,E1 9571.63,E2 9571.63} C_VEL
LIN {X 0,Y 362.597,Z 527.628,A -85,B 0,C 180,E1 9570.845,E2 9570.845} C_VEL
LIN {X 0,Y 365.143,Z 504.202,A -85,B 0,C 180,E1 9570.251,E2 9570.251} C_VEL
LIN {X 0,Y 379.434,Z 301.117,A -85,B 0,C 180,E1 9566.092,E2 9566.092} C_VEL
LIN {X 0,Y 380.257,Z 288.05,A -85,B 0,C 180,E1 9565.796,E2 9565.796} C_VEL
LIN {X 0,Y 372.615,Z 275.657,A -85,B 0,C 180,E1 9562.981,E2 9562.981} C_VEL
LIN {X 0,Y 365.674,Z 265.179,A -85,B 0,C 180,E1 9560.069,E2 9560.069} C_VEL
LIN {X 0,Y 360.081,Z 257.209,A -85,B 0,C 180,E1 9557.367,E2 9557.367} C_VEL
LIN {X 0,Y 356.183,Z 251.932,A -85,B 0,C 180,E1 9555.216,E2 9555.216} C_VEL
LIN {X 0,Y 353.542,Z 248.431,A -85,B 0,C 180,E1 9553.576,E2 9553.576} C_VEL
LIN {X 0,Y 350.201,Z 244.007,A -85,B 0,C 180,E1 9551.195,E2 9551.195} C_VEL
LIN {X 0,Y 346.078,Z 238.835,A -85,B 0,C 180,E1 9547.47,E2 9547.47} C_VEL
LIN {X 0,Y 341.869,Z 234.272,A -85,B 0,C 180,E1 9540.67,E2 9540.67} C_VEL
LIN {X 0,Y 341.371,Z 233.82,A -85,B 0,C 180,E1 9537.65,E2 9537.65} C_VEL
LIN {X 0,Y 341.883,Z 235.677,A -85,B 0,C 180,E1 9533.619,E2 9533.619} C_VEL
LIN {X 0,Y 344.092,Z 238.567,A -85,B 0,C 180,E1 9529.451,E2 9529.451} C_VEL
LIN {X 0,Y 347.695,Z 243.966,A -85,B 0,C 180,E1 9525.426,E2 9525.426} C_VEL
LIN {X 0,Y 351.249,Z 249.394,A -85,B 0,C 180,E1 9522.523,E2 9522.523} C_VEL
LIN {X 0,Y 354.422,Z 254.111,A -85,B 0,C 180,E1 9520.384,E2 9520.384} C_VEL
LIN {X 0,Y 358.788,Z 260.673,A -85,B 0,C 180,E1 9517.857,E2 9517.857} C_VEL
LIN {X 0,Y 364.758,Z 270.109,A -85,B 0,C 180,E1 9514.9,E2 9514.9} C_VEL
LIN {X 0,Y 372.301,Z 282.787,A -85,B 0,C 180,E1 9511.705,E2 9511.705} C_VEL
LIN {X 0,Y 377.945,Z 292.961,A -85,B 0,C 180,E1 9509.586,E2 9509.586} C_VEL
LIN {X 0,Y 363.943,Z 511.487,A -85,B 0,C 180,E1 9505.345,E2 9505.345} C_VEL
LIN {X 0,Y 361.166,Z 535.101,A -85,B 0,C 180,E1 9504.728,E2 9504.728} C_VEL
LIN {X 0,Y 357.644,Z 556.114,A -85,B 0,C 180,E1 9503.962,E2 9503.962} C_VEL
LIN {X 0,Y 353.198,Z 576.395,A -85,B 0,C 180,E1 9502.967,E2 9502.967} C_VEL
LIN {X 0,Y 347.841,Z 596.889,A -85,B 0,C 180,E1 9501.694,E2 9501.694} C_VEL
LIN {X 0,Y 342.073,Z 615.669,A -85,B 0,C 180,E1 9500.238,E2 9500.238} C_VEL
LIN {X 0,Y 335.448,Z 634.609,A -85,B 0,C 180,E1 9498.428,E2 9498.428} C_VEL
LIN {X 0,Y 328.659,Z 652.219,A -85,B 0,C 180,E1 9496.388,E2 9496.388} C_VEL
LIN {X 0,Y 321.556,Z 668.874,A -85,B 0,C 180,E1 9494.022,E2 9494.022} C_VEL
LIN {X 0,Y 314.138,Z 685.198,A -85,B 0,C 180,E1 9491.211,E2 9491.211} C_VEL
LIN {X 0,Y 307.257,Z 699.692,A -85,B 0,C 180,E1 9488.19,E2 9488.19} C_VEL
LIN {X 0,Y 300.695,Z 712.972,A -85,B 0,C 180,E1 9484.783,E2 9484.783} C_VEL
LIN {X 0,Y 294.787,Z 724.974,A -85,B 0,C 180,E1 9481.034,E2 9481.034} C_VEL
LIN {X 0,Y 289.896,Z 735.316,A -85,B 0,C 180,E1 9477.082,E2 9477.082} C_VEL
LIN {X 0,Y 285.947,Z 744.112,A -85,B 0,C 180,E1 9472.837,E2 9472.837} C_VEL
LIN {X 0,Y 283.053,Z 751.491,A -85,B 0,C 180,E1 9468.323,E2 9468.323} C_VEL
LIN {X 0,Y 281.34,Z 756.94,A -85,B 0,C 180,E1 9463.984,E2 9463.984} C_VEL
LIN {X 0,Y 280.437,Z 760.733,A -85,B 0,C 180,E1 9459.646,E2 9459.646} C_VEL
LIN {X 0,Y 280.086,Z 763.204,A -85,B 0,C 180,E1 9455.325,E2 9455.325} C_VEL
LIN {X 0,Y 280.003,Z 764.16,A -85,B 0,C 180,E1 9451.228,E2 9451.228} C_VEL
LIN {X 0,Y 280.018,Z 763.997,A -85,B 0,C 180,E1 9447.135,E2 9447.135} C_VEL
LIN {X 0,Y 280.171,Z 762.45,A -85,B 0,C 180,E1 9443.031,E2 9443.031} C_VEL
LIN {X 0,Y 280.687,Z 759.592,A -85,B 0,C 180,E1 9438.702,E2 9438.702} C_VEL
LIN {X 0,Y 281.852,Z 755.129,A -85,B 0,C 180,E1 9434.36,E2 9434.36} C_VEL
LIN {X 0,Y 284.164,Z 748.53,A -85,B 0,C 180,E1 9429.615,E2 9429.615} C_VEL
LIN {X 0,Y 287.423,Z 740.806,A -85,B 0,C 180,E1 9425.327,E2 9425.327} C_VEL
LIN {X 0,Y 291.861,Z 731.101,A -85,B 0,C 180,E1 9421.117,E2 9421.117} C_VEL
LIN {X 0,Y 297.26,Z 719.993,A -85,B 0,C 180,E1 9417.213,E2 9417.213} C_VEL
LIN {X 0,Y 301.815,Z 710.761,A -85,B 0,C 180,E1 9414.5,E2 9414.5} C_VEL
LIN {X 0,Y 303.073,Z 706.647,A -85,B 0,C 180,E1 9413.277,E2 9413.277} C_VEL
LIN {X 0,Y 303.566,Z 696.231,A -85,B 0,C 180,E1 9410.024,E2 9410.024} C_VEL
LIN {X 0,Y 305.166,Z 691.628,A -85,B 0,C 180,E1 9408.886,E2 9408.886} C_VEL
LIN {X 0,Y 312.499,Z 676.444,A -85,B 0,C 180,E1 9406.03,E2 9406.03} C_VEL
LIN {X 0,Y 320.377,Z 659.14,A -85,B 0,C 180,E1 9403.352,E2 9403.352} C_VEL
LIN {X 0,Y 327.52,Z 642.138,A -85,B 0,C 180,E1 9401.193,E2 9401.193} C_VEL
LIN {X 0,Y 334.505,Z 623.546,A -85,B 0,C 180,E1 9399.272,E2 9399.272} C_VEL
LIN {X 0,Y 341.255,Z 603.333,A -85,B 0,C 180,E1 9397.577,E2 9397.577} C_VEL
LIN {X 0,Y 346.726,Z 584.311,A -85,B 0,C 180,E1 9396.296,E2 9396.296} C_VEL
LIN {X 0,Y 351.721,Z 563.439,A -85,B 0,C 180,E1 9395.185,E2 9395.185} C_VEL
LIN {X 0,Y 355.883,Z 542.002,A -85,B 0,C 180,E1 9394.313,E2 9394.313} C_VEL
LIN {X 0,Y 358.911,Z 520.37,A -85,B 0,C 180,E1 9393.683,E2 9393.683} C_VEL
LIN {X 0,Y 361.3,Z 490.405,A -85,B 0,C 180,E1 9393.05,E2 9393.05} C_VEL
LIN {X 0,Y 374.081,Z 297.272,A -85,B 0,C 180,E1 9389.311,E2 9389.311} C_VEL
LIN {X 0,Y 367.157,Z 284.876,A -85,B 0,C 180,E1 9386.527,E2 9386.527} C_VEL
LIN {X 0,Y 360.677,Z 273.95,A -85,B 0,C 180,E1 9383.528,E2 9383.528} C_VEL
LIN {X 0,Y 354.894,Z 264.656,A -85,B 0,C 180,E1 9380.362,E2 9380.362} C_VEL
LIN {X 0,Y 351.114,Z 258.963,A -85,B 0,C 180,E1 9377.912,E2 9377.912} C_VEL
LIN {X 0,Y 348.282,Z 254.648,A -85,B 0,C 180,E1 9375.741,E2 9375.741} C_VEL
LIN {X 0,Y 345.734,Z 250.644,A -85,B 0,C 180,E1 9373.377,E2 9373.377} C_VEL
LIN {X 0,Y 342.719,Z 245.898,A -85,B 0,C 180,E1 9369.573,E2 9369.573} C_VEL
LIN {X 0,Y 340.599,Z 242.38,A -85,B 0,C 180,E1 9363.198,E2 9363.198} C_VEL
LIN {X 0,Y 340.874,Z 242.296,A -85,B 0,C 180,E1 9360.168,E2 9360.168} C_VEL
LIN {X 0,Y 343.1,Z 245.014,A -85,B 0,C 180,E1 9355.152,E2 9355.152} C_VEL
LIN {X 0,Y 345.414,Z 247.314,A -85,B 0,C 180,E1 9352.348,E2 9352.348} C_VEL
LIN {X 0,Y 349.778,Z 252.94,A -85,B 0,C 180,E1 9348.458,E2 9348.458} C_VEL
LIN {X 0,Y 354.04,Z 258.713,A -85,B 0,C 180,E1 9345.527,E2 9345.527} C_VEL
LIN {X 0,Y 358.188,Z 264.476,A -85,B 0,C 180,E1 9343.124,E2 9343.124} C_VEL
LIN {X 0,Y 364.104,Z 273.131,A -85,B 0,C 180,E1 9340.176,E2 9340.176} C_VEL
LIN {X 0,Y 370.844,Z 283.571,A -85,B 0,C 180,E1 9337.28,E2 9337.28} C_VEL
LIN {X 0,Y 376.352,Z 292.997,A -85,B 0,C 180,E1 9335.155,E2 9335.155} C_VEL
LIN {X 0,Y 361.349,Z 500.21,A -85,B 0,C 180,E1 9330.923,E2 9330.923} C_VEL
LIN {X 0,Y 358.911,Z 523.319,A -85,B 0,C 180,E1 9330.36,E2 9330.36} C_VEL
LIN {X 0,Y 355.046,Z 547.456,A -85,B 0,C 180,E1 9329.559,E2 9329.559} C_VEL
LIN {X 0,Y 350.431,Z 569.943,A -85,B 0,C 180,E1 9328.549,E2 9328.549} C_VEL
LIN {X 0,Y 345.056,Z 590.939,A -85,B 0,C 180,E1 9327.325,E2 9327.325} C_VEL
LIN {X 0,Y 338.664,Z 612.575,A -85,B 0,C 180,E1 9325.755,E2 9325.755} C_VEL
LIN {X 0,Y 331.956,Z 632.5,A -85,B 0,C 180,E1 9323.969,E2 9323.969} C_VEL
LIN {X 0,Y 324.675,Z 651.851,A -85,B 0,C 180,E1 9321.85,E2 9321.85} C_VEL
LIN {X 0,Y 317.234,Z 670.239,A -85,B 0,C 180,E1 9319.426,E2 9319.426} C_VEL
LIN {X 0,Y 309.754,Z 687.305,A -85,B 0,C 180,E1 9316.692,E2 9316.692} C_VEL
LIN {X 0,Y 302.19,Z 703.957,A -85,B 0,C 180,E1 9313.487,E2 9313.487} C_VEL
LIN {X 0,Y 295.313,Z 718.849,A -85,B 0,C 180,E1 9310.037,E2 9310.037} C_VEL
LIN {X 0,Y 289.058,Z 732.277,A -85,B 0,C 180,E1 9306.262,E2 9306.262} C_VEL
LIN {X 0,Y 283.646,Z 744.469,A -85,B 0,C 180,E1 9302.159,E2 9302.159} C_VEL
LIN {X 0,Y 279.392,Z 754.695,A -85,B 0,C 180,E1 9297.956,E2 9297.956} C_VEL
LIN {X 0,Y 275.975,Z 764.039,A -85,B 0,C 180,E1 9293.26,E2 9293.26} C_VEL
LIN {X 0,Y 273.906,Z 770.906,A -85,B 0,C 180,E1 9288.958,E2 9288.958} C_VEL
LIN {X 0,Y 272.61,Z 776.74,A -85,B 0,C 180,E1 9284.225,E2 9284.225} C_VEL
LIN {X 0,Y 272.109,Z 780.429,A -85,B 0,C 180,E1 9280.158,E2 9280.158} C_VEL
LIN {X 0,Y 271.968,Z 783.107,A -85,B 0,C 180,E1 9275.697,E2 9275.697} C_VEL
LIN {X 0,Y 271.981,Z 784.178,A -85,B 0,C 180,E1 9271.685,E2 9271.685} C_VEL
LIN {X 0,Y 271.981,Z 784.152,A -85,B 0,C 180,E1 9268.104,E2 9268.104} C_VEL
LIN {X 0,Y 271.978,Z 782.947,A -85,B 0,C 180,E1 9263.88,E2 9263.88} C_VEL
LIN {X 0,Y 272.125,Z 780.251,A -85,B 0,C 180,E1 9259.628,E2 9259.628} C_VEL
LIN {X 0,Y 272.668,Z 776.431,A -85,B 0,C 180,E1 9255.482,E2 9255.482} C_VEL
LIN {X 0,Y 274.075,Z 770.252,A -85,B 0,C 180,E1 9250.612,E2 9250.612} C_VEL
LIN {X 0,Y 276.369,Z 762.905,A -85,B 0,C 180,E1 9246.097,E2 9246.097} C_VEL
LIN {X 0,Y 279.865,Z 753.453,A -85,B 0,C 180,E1 9241.506,E2 9241.506} C_VEL
LIN {X 0,Y 284.476,Z 742.521,A -85,B 0,C 180,E1 9237.142,E2 9237.142} C_VEL
LIN {X 0,Y 289.659,Z 730.917,A -85,B 0,C 180,E1 9233.334,E2 9233.334} C_VEL
LIN {X 0,Y 296.378,Z 716.402,A -85,B 0,C 180,E1 9229.377,E2 9229.377} C_VEL
LIN {X 0,Y 303.558,Z 700.991,A -85,B 0,C 180,E1 9225.893,E2 9225.893} C_VEL
LIN {X 0,Y 310.933,Z 684.555,A -85,B 0,C 180,E1 9222.849,E2 9222.849} C_VEL
LIN {X 0,Y 318.885,Z 666.038,A -85,B 0,C 180,E1 9219.999,E2 9219.999} C_VEL
LIN {X 0,Y 326.085,Z 648.124,A -85,B 0,C 180,E1 9217.714,E2 9217.714} C_VEL
LIN {X 0,Y 333.073,Z 629.029,A -85,B 0,C 180,E1 9215.709,E2 9215.709} C_VEL
LIN {X 0,Y 339.854,Z 608.656,A -85,B 0,C 180,E1 9213.94,E2 9213.94} C_VEL
LIN {X 0,Y 345.631,Z 588.531,A -85,B 0,C 180,E1 9212.531,E2 9212.531} C_VEL
LIN {X 0,Y 351.208,Z 565.953,A -85,B 0,C 180,E1 9211.267,E2 9211.267} C_VEL
LIN {X 0,Y 355.588,Z 544.147,A -85,B 0,C 180,E1 9210.321,E2 9210.321} C_VEL
LIN {X 0,Y 359.098,Z 521.151,A -85,B 0,C 180,E1 9209.592,E2 9209.592} C_VEL
LIN {X 0,Y 361.506,Z 496.806,A -85,B 0,C 180,E1 9209.015,E2 9209.015} C_VEL
LIN {X 0,Y 376.27,Z 292.744,A -85,B 0,C 180,E1 9204.846,E2 9204.846} C_VEL
LIN {X 0,Y 369.752,Z 281.97,A -85,B 0,C 180,E1 9202.329,E2 9202.329} C_VEL
LIN {X 0,Y 363.341,Z 272.049,A -85,B 0,C 180,E1 9199.533,E2 9199.533} C_VEL
LIN {X 0,Y 357.905,Z 264.158,A -85,B 0,C 180,E1 9196.806,E2 9196.806} C_VEL
LIN {X 0,Y 352.792,Z 256.927,A -85,B 0,C 180,E1 9193.772,E2 9193.772} C_VEL
LIN {X 0,Y 348.791,Z 251.698,A -85,B 0,C 180,E1 9190.906,E2 9190.906} C_VEL
LIN {X 0,Y 344.783,Z 246.586,A -85,B 0,C 180,E1 9187.163,E2 9187.163} C_VEL
LIN {X 0,Y 340.845,Z 242.157,A -85,B 0,C 180,E1 9180.504,E2 9180.504} C_VEL
LIN {X 0,Y 340.396,Z 241.767,A -85,B 0,C 180,E1 9177.643,E2 9177.643} C_VEL
LIN {X 0,Y 340.964,Z 243.777,A -85,B 0,C 180,E1 9173.433,E2 9173.433} C_VEL
LIN {X 0,Y 342.954,Z 246.398,A -85,B 0,C 180,E1 9169.671,E2 9169.671} C_VEL
LIN {X 0,Y 346.379,Z 251.687,A -85,B 0,C 180,E1 9165.711,E2 9165.711} C_VEL
LIN {X 0,Y 349.742,Z 256.956,A -85,B 0,C 180,E1 9162.875,E2 9162.875} C_VEL
LIN {X 0,Y 352.893,Z 261.795,A -85,B 0,C 180,E1 9160.683,E2 9160.683} C_VEL
LIN {X 0,Y 357.253,Z 268.475,A -85,B 0,C 180,E1 9158.103,E2 9158.103} C_VEL
LIN {X 0,Y 363.046,Z 277.982,A -85,B 0,C 180,E1 9155.165,E2 9155.165} C_VEL
LIN {X 0,Y 370.212,Z 290.323,A -85,B 0,C 180,E1 9152.057,E2 9152.057} C_VEL
LIN {X 0,Y 373.955,Z 297.462,A -85,B 0,C 180,E1 9150.583,E2 9150.583} C_VEL
LIN {X 0,Y 359.533,Z 513.598,A -85,B 0,C 180,E1 9146.378,E2 9146.378} C_VEL
LIN {X 0,Y 356.689,Z 536.132,A -85,B 0,C 180,E1 9145.775,E2 9145.775} C_VEL
LIN {X 0,Y 353.027,Z 557.036,A -85,B 0,C 180,E1 9145.005,E2 9145.005} C_VEL
LIN {X 0,Y 348.458,Z 577.168,A -85,B 0,C 180,E1 9144.012,E2 9144.012} C_VEL
LIN {X 0,Y 342.638,Z 598.495,A -85,B 0,C 180,E1 9142.671,E2 9142.671} C_VEL
LIN {X 0,Y 336.425,Z 618.002,A -85,B 0,C 180,E1 9141.137,E2 9141.137} C_VEL
LIN {X 0,Y 329.603,Z 636.532,A -85,B 0,C 180,E1 9139.32,E2 9139.32} C_VEL
LIN {X 0,Y 322.083,Z 655.024,A -85,B 0,C 180,E1 9137.105,E2 9137.105} C_VEL
LIN {X 0,Y 314.572,Z 671.989,A -85,B 0,C 180,E1 9134.622,E2 9134.622} C_VEL
LIN {X 0,Y 307.174,Z 687.372,A -85,B 0,C 180,E1 9131.856,E2 9131.856} C_VEL
LIN {X 0,Y 299.689,Z 702.289,A -85,B 0,C 180,E1 9128.6,E2 9128.6} C_VEL
LIN {X 0,Y 293.141,Z 715.053,A -85,B 0,C 180,E1 9125.199,E2 9125.199} C_VEL
LIN {X 0,Y 287.219,Z 726.414,A -85,B 0,C 180,E1 9121.473,E2 9121.473} C_VEL
LIN {X 0,Y 281.943,Z 736.954,A -85,B 0,C 180,E1 9117.223,E2 9117.223} C_VEL
LIN {X 0,Y 277.931,Z 745.586,A -85,B 0,C 180,E1 9112.862,E2 9112.862} C_VEL
LIN {X 0,Y 275.103,Z 752.371,A -85,B 0,C 180,E1 9108.433,E2 9108.433} C_VEL
LIN {X 0,Y 273.281,Z 757.841,A -85,B 0,C 180,E1 9103.757,E2 9103.757} C_VEL
LIN {X 0,Y 272.428,Z 761.33,A -85,B 0,C 180,E1 9099.506,E2 9099.506} C_VEL
LIN {X 0,Y 272.082,Z 763.622,A -85,B 0,C 180,E1 9095.06,E2 9095.06} C_VEL
LIN {X 0,Y 272.009,Z 764.472,A -85,B 0,C 180,E1 9091.053,E2 9091.053} C_VEL
LIN {X 0,Y 272.034,Z 764.164,A -85,B 0,C 180,E1 9086.629,E2 9086.629} C_VEL
LIN {X 0,Y 272.225,Z 762.53,A -85,B 0,C 180,E1 9082.402,E2 9082.402} C_VEL
LIN {X 0,Y 272.889,Z 759.304,A -85,B 0,C 180,E1 9077.731,E2 9077.731} C_VEL
LIN {X 0,Y 274.286,Z 754.705,A -85,B 0,C 180,E1 9073.263,E2 9073.263} C_VEL
LIN {X 0,Y 276.799,Z 748.16,A -85,B 0,C 180,E1 9068.603,E2 9068.603} C_VEL
LIN {X 0,Y 280.396,Z 740.246,A -85,B 0,C 180,E1 9064.213,E2 9064.213} C_VEL
LIN {X 0,Y 285.074,Z 730.714,A -85,B 0,C 180,E1 9060.034,E2 9060.034} C_VEL
LIN {X 0,Y 290.718,Z 719.704,A -85,B 0,C 180,E1 9056.141,E2 9056.141} C_VEL
LIN {X 0,Y 297.279,Z 707.127,A -85,B 0,C 180,E1 9052.501,E2 9052.501} C_VEL
LIN {X 0,Y 304.014,Z 693.851,A -85,B 0,C 180,E1 9049.37,E2 9049.37} C_VEL
LIN {X 0,Y 305.166,Z 691.628,A -85,B 0,C 180,E1 9048.886,E2 9048.886} C_VEL
LIN {X 0,Y 306.853,Z 686.911,A -85,B 0,C 180,E1 9047.774,E2 9047.774} C_VEL
LIN {X 0,Y 308.393,Z 674.937,A -85,B 0,C 180,E1 9044.775,E2 9044.775} C_VEL
LIN {X 0,Y 310.187,Z 669.623,A -85,B 0,C 180,E1 9043.782,E2 9043.782} C_VEL
LIN {X 0,Y 317.837,Z 652.984,A -85,B 0,C 180,E1 9041.387,E2 9041.387} C_VEL
LIN {X 0,Y 325.294,Z 635.006,A -85,B 0,C 180,E1 9039.286,E2 9039.286} C_VEL
LIN {X 0,Y 332.478,Z 615.769,A -85,B 0,C 180,E1 9037.448,E2 9037.448} C_VEL
LIN {X 0,Y 338.7,Z 596.691,A -85,B 0,C 180,E1 9035.977,E2 9035.977} C_VEL
LIN {X 0,Y 344.475,Z 575.754,A -85,B 0,C 180,E1 9034.693,E2 9034.693} C_VEL
LIN {X 0,Y 349.198,Z 555.193,A -85,B 0,C 180,E1 9033.705,E2 9033.705} C_VEL
LIN {X 0,Y 352.912,Z 534.139,A -85,B 0,C 180,E1 9032.956,E2 9032.956} C_VEL
LIN {X 0,Y 355.778,Z 510.642,A -85,B 0,C 180,E1 9032.355,E2 9032.355} C_VEL
LIN {X 0,Y 370.207,Z 301.675,A -85,B 0,C 180,E1 9028.286,E2 9028.286} C_VEL
LIN {X 0,Y 364.217,Z 290.811,A -85,B 0,C 180,E1 9025.749,E2 9025.749} C_VEL
LIN {X 0,Y 358.139,Z 280.189,A -85,B 0,C 180,E1 9022.791,E2 9022.791} C_VEL
LIN {X 0,Y 352.634,Z 271.333,A -85,B 0,C 180,E1 9019.633,E2 9019.633} C_VEL
LIN {X 0,Y 349.362,Z 266.201,A -85,B 0,C 180,E1 9017.402,E2 9017.402} C_VEL
LIN {X 0,Y 346.832,Z 262.215,A -85,B 0,C 180,E1 9015.38,E2 9015.38} C_VEL
LIN {X 0,Y 344.445,Z 258.36,A -85,B 0,C 180,E1 9013.087,E2 9013.087} C_VEL
LIN {X 0,Y 341.542,Z 253.691,A -85,B 0,C 180,E1 9009.266,E2 9009.266} C_VEL
LIN {X 0,Y 339.62,Z 250.283,A -85,B 0,C 180,E1 9003.038,E2 9003.038} C_VEL
LIN {X 0,Y 339.935,Z 250.286,A -85,B 0,C 180,E1 9000,E2 9000} C_VEL
LIN {X 0,Y 342.598,Z 253.47,A -85,B 0,C 180,E1 8994.474,E2 8994.474} C_VEL
LIN {X 0,Y 344.267,Z 255.245,A -85,B 0,C 180,E1 8992.491,E2 8992.491} C_VEL
LIN {X 0,Y 348.362,Z 260.629,A -85,B 0,C 180,E1 8988.746,E2 8988.746} C_VEL
LIN {X 0,Y 352.525,Z 266.421,A -85,B 0,C 180,E1 8985.798,E2 8985.798} C_VEL
LIN {X 0,Y 356.879,Z 272.604,A -85,B 0,C 180,E1 8983.228,E2 8983.228} C_VEL
LIN {X 0,Y 363.147,Z 282.006,A -85,B 0,C 180,E1 8980.079,E2 8980.079} C_VEL
LIN {X 0,Y 370.67,Z 294.298,A -85,B 0,C 180,E1 8976.85,E2 8976.85} C_VEL
LIN {X 0,Y 372.4,Z 297.477,A -85,B 0,C 180,E1 8976.162,E2 8976.162} C_VEL
LIN {X 0,Y 357.031,Z 502.568,A -85,B 0,C 180,E1 8971.969,E2 8971.969} C_VEL
LIN {X 0,Y 354.532,Z 524.987,A -85,B 0,C 180,E1 8971.416,E2 8971.416} C_VEL
LIN {X 0,Y 350.657,Z 548.117,A -85,B 0,C 180,E1 8970.64,E2 8970.64} C_VEL
LIN {X 0,Y 345.87,Z 570.602,A -85,B 0,C 180,E1 8969.627,E2 8969.627} C_VEL
LIN {X 0,Y 340.377,Z 591.401,A -85,B 0,C 180,E1 8968.413,E2 8968.413} C_VEL
LIN {X 0,Y 333.481,Z 613.843,A -85,B 0,C 180,E1 8966.771,E2 8966.771} C_VEL
LIN {X 0,Y 326.576,Z 633.631,A -85,B 0,C 180,E1 8964.981,E2 8964.981} C_VEL
LIN {X 0,Y 319.19,Z 652.431,A -85,B 0,C 180,E1 8962.895,E2 8962.895} C_VEL
LIN {X 0,Y 311.354,Z 670.971,A -85,B 0,C 180,E1 8960.416,E2 8960.416} C_VEL
LIN {X 0,Y 303.871,Z 687.371,A -85,B 0,C 180,E1 8957.759,E2 8957.759} C_VEL
LIN {X 0,Y 295.73,Z 704.464,A -85,B 0,C 180,E1 8954.415,E2 8954.415} C_VEL
LIN {X 0,Y 288.559,Z 719.285,A -85,B 0,C 180,E1 8950.91,E2 8950.91} C_VEL
LIN {X 0,Y 282.006,Z 732.596,A -85,B 0,C 180,E1 8947.065,E2 8947.065} C_VEL
LIN {X 0,Y 276.063,Z 745.216,A -85,B 0,C 180,E1 8942.659,E2 8942.659} C_VEL
LIN {X 0,Y 271.641,Z 755.331,A -85,B 0,C 180,E1 8938.347,E2 8938.347} C_VEL
LIN {X 0,Y 268.218,Z 764.098,A -85,B 0,C 180,E1 8933.74,E2 8933.74} C_VEL
LIN {X 0,Y 266.024,Z 770.917,A -85,B 0,C 180,E1 8929.314,E2 8929.314} C_VEL
LIN {X 0,Y 264.645,Z 776.659,A -85,B 0,C 180,E1 8924.439,E2 8924.439} C_VEL
LIN {X 0,Y 264.11,Z 780.364,A -85,B 0,C 180,E1 8920.168,E2 8920.168} C_VEL
LIN {X 0,Y 263.971,Z 782.889,A -85,B 0,C 180,E1 8915.652,E2 8915.652} C_VEL
LIN {X 0,Y 263.986,Z 783.887,A -85,B 0,C 180,E1 8911.736,E2 8911.736} C_VEL
LIN {X 0,Y 263.986,Z 783.861,A -85,B 0,C 180,E1 8908.047,E2 8908.047} C_VEL
LIN {X 0,Y 263.985,Z 782.654,A -85,B 0,C 180,E1 8903.694,E2 8903.694} C_VEL
LIN {X 0,Y 264.152,Z 779.953,A -85,B 0,C 180,E1 8899.312,E2 8899.312} C_VEL
LIN {X 0,Y 264.734,Z 776.209,A -85,B 0,C 180,E1 8895.119,E2 8895.119} C_VEL
LIN {X 0,Y 266.202,Z 770.261,A -85,B 0,C 180,E1 8890.243,E2 8890.243} C_VEL
LIN {X 0,Y 268.491,Z 763.332,A -85,B 0,C 180,E1 8885.819,E2 8885.819} C_VEL
LIN {X 0,Y 272.223,Z 753.865,A -85,B 0,C 180,E1 8881,E2 8881} C_VEL
LIN {X 0,Y 276.835,Z 743.575,A -85,B 0,C 180,E1 8876.704,E2 8876.704} C_VEL
LIN {X 0,Y 282.635,Z 731.233,A -85,B 0,C 180,E1 8872.522,E2 8872.522} C_VEL
LIN {X 0,Y 289.669,Z 716.838,A -85,B 0,C 180,E1 8868.493,E2 8868.493} C_VEL
LIN {X 0,Y 296.58,Z 702.648,A -85,B 0,C 180,E1 8865.204,E2 8865.204} C_VEL
LIN {X 0,Y 304.34,Z 686.238,A -85,B 0,C 180,E1 8862.058,E2 8862.058} C_VEL
LIN {X 0,Y 312.098,Z 669.183,A -85,B 0,C 180,E1 8859.33,E2 8859.33} C_VEL
LIN {X 0,Y 319.669,Z 651.073,A -85,B 0,C 180,E1 8856.953,E2 8856.953} C_VEL
LIN {X 0,Y 327.636,Z 630.401,A -85,B 0,C 180,E1 8854.719,E2 8854.719} C_VEL
LIN {X 0,Y 334.627,Z 610.233,A -85,B 0,C 180,E1 8852.943,E2 8852.943} C_VEL
LIN {X 0,Y 340.8,Z 589.581,A -85,B 0,C 180,E1 8851.481,E2 8851.481} C_VEL
LIN {X 0,Y 346.379,Z 568.034,A -85,B 0,C 180,E1 8850.255,E2 8850.255} C_VEL
LIN {X 0,Y 351.007,Z 545.825,A -85,B 0,C 180,E1 8849.28,E2 8849.28} C_VEL
LIN {X 0,Y 354.828,Z 521.972,A -85,B 0,C 180,E1 8848.513,E2 8848.513} C_VEL
LIN {X 0,Y 357.29,Z 498.397,A -85,B 0,C 180,E1 8847.949,E2 8847.949} C_VEL
LIN {X 0,Y 372.307,Z 297.19,A -85,B 0,C 180,E1 8843.84,E2 8843.84} C_VEL
LIN {X 0,Y 365.161,Z 285.335,A -85,B 0,C 180,E1 8840.894,E2 8840.894} C_VEL
LIN {X 0,Y 358.979,Z 275.858,A -85,B 0,C 180,E1 8837.967,E2 8837.967} C_VEL
LIN {X 0,Y 354.028,Z 268.553,A -85,B 0,C 180,E1 8835.227,E2 8835.227} C_VEL
LIN {X 0,Y 350.353,Z 263.5,A -85,B 0,C 180,E1 8832.862,E2 8832.862} C_VEL
LIN {X 0,Y 347.391,Z 259.388,A -85,B 0,C 180,E1 8830.614,E2 8830.614} C_VEL
LIN {X 0,Y 343.498,Z 254.334,A -85,B 0,C 180,E1 8826.854,E2 8826.854} C_VEL
LIN {X 0,Y 339.823,Z 250.047,A -85,B 0,C 180,E1 8820.337,E2 8820.337} C_VEL
LIN {X 0,Y 339.414,Z 249.755,A -85,B 0,C 180,E1 8817.467,E2 8817.467} C_VEL
LIN {X 0,Y 340.312,Z 252.282,A -85,B 0,C 180,E1 8812.572,E2 8812.572} C_VEL
LIN {X 0,Y 341.814,Z 254.227,A -85,B 0,C 180,E1 8809.891,E2 8809.891} C_VEL
LIN {X 0,Y 345.153,Z 259.562,A -85,B 0,C 180,E1 8805.916,E2 8805.916} C_VEL
LIN {X 0,Y 348.347,Z 264.694,A -85,B 0,C 180,E1 8803.148,E2 8803.148} C_VEL
LIN {X 0,Y 351.258,Z 269.274,A -85,B 0,C 180,E1 8801.064,E2 8801.064} C_VEL
LIN {X 0,Y 355.515,Z 275.958,A -85,B 0,C 180,E1 8798.468,E2 8798.468} C_VEL
LIN {X 0,Y 361.419,Z 285.966,A -85,B 0,C 180,E1 8795.395,E2 8795.395} C_VEL
LIN {X 0,Y 367.953,Z 297.582,A -85,B 0,C 180,E1 8792.487,E2 8792.487} C_VEL
LIN {X 0,Y 370.078,Z 301.943,A -85,B 0,C 180,E1 8791.604,E2 8791.604} C_VEL
LIN {X 0,Y 355.386,Z 514.02,A -85,B 0,C 180,E1 8787.473,E2 8787.473} C_VEL
LIN {X 0,Y 352.455,Z 536.38,A -85,B 0,C 180,E1 8786.873,E2 8786.873} C_VEL
LIN {X 0,Y 348.693,Z 557.19,A -85,B 0,C 180,E1 8786.109,E2 8786.109} C_VEL
LIN {X 0,Y 344.051,Z 577.076,A -85,B 0,C 180,E1 8785.134,E2 8785.134} C_VEL
LIN {X 0,Y 338.161,Z 598.111,A -85,B 0,C 180,E1 8783.82,E2 8783.82} C_VEL
LIN {X 0,Y 332.045,Z 616.779,A -85,B 0,C 180,E1 8782.366,E2 8782.366} C_VEL
LIN {X 0,Y 324.99,Z 635.555,A -85,B 0,C 180,E1 8780.552,E2 8780.552} C_VEL
LIN {X 0,Y 317.451,Z 653.651,A -85,B 0,C 180,E1 8778.419,E2 8778.419} C_VEL
LIN {X 0,Y 309.845,Z 670.215,A -85,B 0,C 180,E1 8776.021,E2 8776.021} C_VEL
LIN {X 0,Y 302.08,Z 685.929,A -85,B 0,C 180,E1 8773.246,E2 8773.246} C_VEL
LIN {X 0,Y 294.602,Z 700.383,A -85,B 0,C 180,E1 8770.153,E2 8770.153} C_VEL
LIN {X 0,Y 287.559,Z 713.351,A -85,B 0,C 180,E1 8766.729,E2 8766.729} C_VEL
LIN {X 0,Y 280.871,Z 725.617,A -85,B 0,C 180,E1 8762.757,E2 8762.757} C_VEL
LIN {X 0,Y 275.404,Z 735.943,A -85,B 0,C 180,E1 8758.634,E2 8758.634} C_VEL
LIN {X 0,Y 270.94,Z 744.731,A -85,B 0,C 180,E1 8754.181,E2 8754.181} C_VEL
LIN {X 0,Y 267.615,Z 752.097,A -85,B 0,C 180,E1 8749.421,E2 8749.421} C_VEL
LIN {X 0,Y 265.617,Z 757.54,A -85,B 0,C 180,E1 8744.831,E2 8744.831} C_VEL
LIN {X 0,Y 264.545,Z 761.324,A -85,B 0,C 180,E1 8740.232,E2 8740.232} C_VEL
LIN {X 0,Y 264.114,Z 763.788,A -85,B 0,C 180,E1 8735.649,E2 8735.649} C_VEL
LIN {X 0,Y 264.013,Z 764.72,A -85,B 0,C 180,E1 8731.519,E2 8731.519} C_VEL
LIN {X 0,Y 264.024,Z 764.627,A -85,B 0,C 180,E1 8727.395,E2 8727.395} C_VEL
LIN {X 0,Y 264.202,Z 763.142,A -85,B 0,C 180,E1 8722.826,E2 8722.826} C_VEL
LIN {X 0,Y 264.752,Z 760.496,A -85,B 0,C 180,E1 8718.454,E2 8718.454} C_VEL
LIN {X 0,Y 266.048,Z 756.209,A -85,B 0,C 180,E1 8713.853,E2 8713.853} C_VEL
LIN {X 0,Y 268.347,Z 750.48,A -85,B 0,C 180,E1 8709.265,E2 8709.265} C_VEL
LIN {X 0,Y 271.808,Z 742.975,A -85,B 0,C 180,E1 8704.742,E2 8704.742} C_VEL
LIN {X 0,Y 276.832,Z 733.192,A -85,B 0,C 180,E1 8700.093,E2 8700.093} C_VEL
LIN {X 0,Y 282.651,Z 722.486,A -85,B 0,C 180,E1 8696.02,E2 8696.02} C_VEL
LIN {X 0,Y 289.292,Z 710.261,A -85,B 0,C 180,E1 8692.285,E2 8692.285} C_VEL
LIN {X 0,Y 296.572,Z 696.669,A -85,B 0,C 180,E1 8688.898,E2 8688.898} C_VEL
LIN {X 0,Y 304.283,Z 681.771,A -85,B 0,C 180,E1 8685.845,E2 8685.845} C_VEL
LIN {X 0,Y 310.187,Z 669.623,A -85,B 0,C 180,E1 8683.782,E2 8683.782} C_VEL
LIN {X 0,Y 312.037,Z 664.31,A -85,B 0,C 180,E1 8682.815,E2 8682.815} C_VEL
LIN {X 0,Y 314.281,Z 650.928,A -85,B 0,C 180,E1 8680.101,E2 8680.101} C_VEL
LIN {X 0,Y 316.237,Z 645.001,A -85,B 0,C 180,E1 8679.238,E2 8679.238} C_VEL
LIN {X 0,Y 324.266,Z 625.34,A -85,B 0,C 180,E1 8677.151,E2 8677.151} C_VEL
LIN {X 0,Y 331.11,Z 606.503,A -85,B 0,C 180,E1 8675.532,E2 8675.532} C_VEL
LIN {X 0,Y 337.194,Z 586.757,A -85,B 0,C 180,E1 8674.18,E2 8674.18} C_VEL
LIN {X 0,Y 342.796,Z 565.202,A -85,B 0,C 180,E1 8673.013,E2 8673.013} C_VEL
LIN {X 0,Y 347.285,Z 543.74,A -85,B 0,C 180,E1 8672.131,E2 8672.131} C_VEL
LIN {X 0,Y 350.605,Z 521.81,A -85,B 0,C 180,E1 8671.486,E2 8671.486} C_VEL
LIN {X 0,Y 353.118,Z 493.754,A -85,B 0,C 180,E1 8670.881,E2 8670.881} C_VEL
LIN {X 0,Y 366.439,Z 306.149,A -85,B 0,C 180,E1 8667.24,E2 8667.24} C_VEL
LIN {X 0,Y 360.94,Z 295.992,A -85,B 0,C 180,E1 8664.771,E2 8664.771} C_VEL
LIN {X 0,Y 355.708,Z 286.691,A -85,B 0,C 180,E1 8662.084,E2 8662.084} C_VEL
LIN {X 0,Y 350.921,Z 278.714,A -85,B 0,C 180,E1 8659.214,E2 8659.214} C_VEL
LIN {X 0,Y 347.748,Z 273.597,A -85,B 0,C 180,E1 8656.968,E2 8656.968} C_VEL
LIN {X 0,Y 345.301,Z 269.645,A -85,B 0,C 180,E1 8654.934,E2 8654.934} C_VEL
LIN {X 0,Y 343.165,Z 266.075,A -85,B 0,C 180,E1 8652.794,E2 8652.794} C_VEL
LIN {X 0,Y 340.476,Z 261.577,A -85,B 0,C 180,E1 8649.125,E2 8649.125} C_VEL
LIN {X 0,Y 338.644,Z 258.236,A -85,B 0,C 180,E1 8643.047,E2 8643.047} C_VEL
LIN {X 0,Y 338.943,Z 258.211,A -85,B 0,C 180,E1 8640.077,E2 8640.077} C_VEL
LIN {X 0,Y 341.616,Z 261.459,A -85,B 0,C 180,E1 8634.458,E2 8634.458} C_VEL
LIN {X 0,Y 343.121,Z 263.171,A -85,B 0,C 180,E1 8632.634,E2 8632.634} C_VEL
LIN {X 0,Y 347.047,Z 268.477,A -85,B 0,C 180,E1 8628.955,E2 8628.955} C_VEL
LIN {X 0,Y 350.898,Z 273.949,A -85,B 0,C 180,E1 8626.152,E2 8626.152} C_VEL
LIN {X 0,Y 355.715,Z 280.909,A -85,B 0,C 180,E1 8623.255,E2 8623.255} C_VEL
LIN {X 0,Y 361.84,Z 290.618,A -85,B 0,C 180,E1 8620.131,E2 8620.131} C_VEL
LIN {X 0,Y 368.416,Z 301.637,A -85,B 0,C 180,E1 8617.249,E2 8617.249} C_VEL
LIN {X 0,Y 368.504,Z 302.604,A -85,B 0,C 180,E1 8617.175,E2 8617.175} C_VEL
LIN {X 0,Y 352.88,Z 504.49,A -85,B 0,C 180,E1 8613.05,E2 8613.05} C_VEL
LIN {X 0,Y 350.132,Z 527.786,A -85,B 0,C 180,E1 8612.467,E2 8612.467} C_VEL
LIN {X 0,Y 346.079,Z 550.397,A -85,B 0,C 180,E1 8611.683,E2 8611.683} C_VEL
LIN {X 0,Y 340.825,Z 573.595,A -85,B 0,C 180,E1 8610.606,E2 8610.606} C_VEL
LIN {X 0,Y 334.853,Z 595.296,A -85,B 0,C 180,E1 8609.309,E2 8609.309} C_VEL
LIN {X 0,Y 328.124,Z 615.938,A -85,B 0,C 180,E1 8607.75,E2 8607.75} C_VEL
LIN {X 0,Y 320.633,Z 636.372,A -85,B 0,C 180,E1 8605.854,E2 8605.854} C_VEL
LIN {X 0,Y 313.075,Z 654.786,A -85,B 0,C 180,E1 8603.759,E2 8603.759} C_VEL
LIN {X 0,Y 304.851,Z 673.222,A -85,B 0,C 180,E1 8601.212,E2 8601.212} C_VEL
LIN {X 0,Y 296.835,Z 690.101,A -85,B 0,C 180,E1 8598.397,E2 8598.397} C_VEL
LIN {X 0,Y 288.91,Z 705.84,A -85,B 0,C 180,E1 8595.19,E2 8595.19} C_VEL
LIN {X 0,Y 281.091,Z 721.133,A -85,B 0,C 180,E1 8591.422,E2 8591.422} C_VEL
LIN {X 0,Y 274.686,Z 733.575,A -85,B 0,C 180,E1 8587.698,E2 8587.698} C_VEL
LIN {X 0,Y 268.502,Z 745.963,A -85,B 0,C 180,E1 8583.188,E2 8583.188} C_VEL
LIN {X 0,Y 263.703,Z 756.423,A -85,B 0,C 180,E1 8578.537,E2 8578.537} C_VEL
LIN {X 0,Y 260.196,Z 764.899,A -85,B 0,C 180,E1 8573.796,E2 8573.796} C_VEL
LIN {X 0,Y 257.801,Z 772.071,A -85,B 0,C 180,E1 8568.778,E2 8568.778} C_VEL
LIN {X 0,Y 256.595,Z 777.016,A -85,B 0,C 180,E1 8564.21,E2 8564.21} C_VEL
LIN {X 0,Y 256.066,Z 780.793,A -85,B 0,C 180,E1 8559.439,E2 8559.439} C_VEL
LIN {X 0,Y 255.975,Z 782.835,A -85,B 0,C 180,E1 8555.097,E2 8555.097} C_VEL
LIN {X 0,Y 255.996,Z 783.645,A -85,B 0,C 180,E1 8551.343,E2 8551.343} C_VEL
LIN {X 0,Y 255.988,Z 783.496,A -85,B 0,C 180,E1 8547.314,E2 8547.314} C_VEL
LIN {X 0,Y 256.005,Z 781.967,A -85,B 0,C 180,E1 8542.757,E2 8542.757} C_VEL
LIN {X 0,Y 256.227,Z 779.315,A -85,B 0,C 180,E1 8538.521,E2 8538.521} C_VEL
LIN {X 0,Y 257.039,Z 775.01,A -85,B 0,C 180,E1 8533.736,E2 8533.736} C_VEL
LIN {X 0,Y 258.736,Z 768.993,A -85,B 0,C 180,E1 8528.938,E2 8528.938} C_VEL
LIN {X 0,Y 261.706,Z 761.058,A -85,B 0,C 180,E1 8523.938,E2 8523.938} C_VEL
LIN {X 0,Y 265.59,Z 752.106,A -85,B 0,C 180,E1 8519.455,E2 8519.455} C_VEL
LIN {X 0,Y 271.267,Z 740.283,A -85,B 0,C 180,E1 8514.643,E2 8514.643} C_VEL
LIN {X 0,Y 277.768,Z 727.587,A -85,B 0,C 180,E1 8510.423,E2 8510.423} C_VEL
LIN {X 0,Y 285.062,Z 713.3,A -85,B 0,C 180,E1 8506.571,E2 8506.571} C_VEL
LIN {X 0,Y 293.462,Z 696.721,A -85,B 0,C 180,E1 8502.903,E2 8502.903} C_VEL
LIN {X 0,Y 301.598,Z 680.109,A -85,B 0,C 180,E1 8499.875,E2 8499.875} C_VEL
LIN {X 0,Y 309.547,Z 662.671,A -85,B 0,C 180,E1 8497.283,E2 8497.283} C_VEL
LIN {X 0,Y 317.982,Z 642.796,A -85,B 0,C 180,E1 8494.849,E2 8494.849} C_VEL
LIN {X 0,Y 325.27,Z 623.854,A -85,B 0,C 180,E1 8492.949,E2 8492.949} C_VEL
LIN {X 0,Y 332.241,Z 603.329,A -85,B 0,C 180,E1 8491.278,E2 8491.278} C_VEL
LIN {X 0,Y 338.443,Z 582.531,A -85,B 0,C 180,E1 8489.902,E2 8489.902} C_VEL
LIN {X 0,Y 343.529,Z 561.924,A -85,B 0,C 180,E1 8488.83,E2 8488.83} C_VEL
LIN {X 0,Y 348.14,Z 539.148,A -85,B 0,C 180,E1 8487.911,E2 8487.911} C_VEL
LIN {X 0,Y 351.399,Z 517.519,A -85,B 0,C 180,E1 8487.269,E2 8487.269} C_VEL
LIN {X 0,Y 354.28,Z 485.73,A -85,B 0,C 180,E1 8486.563,E2 8486.563} C_VEL
LIN {X 0,Y 368.449,Z 301.802,A -85,B 0,C 180,E1 8482.812,E2 8482.812} C_VEL
LIN {X 0,Y 362.044,Z 291.046,A -85,B 0,C 180,E1 8480.026,E2 8480.026} C_VEL
LIN {X 0,Y 356.486,Z 282.302,A -85,B 0,C 180,E1 8477.253,E2 8477.253} C_VEL
LIN {X 0,Y 351.726,Z 275.214,A -85,B 0,C 180,E1 8474.487,E2 8474.487} C_VEL
LIN {X 0,Y 348.555,Z 270.742,A -85,B 0,C 180,E1 8472.34,E2 8472.34} C_VEL
LIN {X 0,Y 345.901,Z 266.978,A -85,B 0,C 180,E1 8470.24,E2 8470.24} C_VEL
LIN {X 0,Y 342.369,Z 262.206,A -85,B 0,C 180,E1 8466.708,E2 8466.708} C_VEL
LIN {X 0,Y 338.804,Z 257.94,A -85,B 0,C 180,E1 8460.169,E2 8460.169} C_VEL
LIN {X 0,Y 338.438,Z 257.707,A -85,B 0,C 180,E1 8457.46,E2 8457.46} C_VEL
LIN {X 0,Y 339.343,Z 260.283,A -85,B 0,C 180,E1 8452.551,E2 8452.551} C_VEL
LIN {X 0,Y 340.679,Z 262.053,A -85,B 0,C 180,E1 8450.114,E2 8450.114} C_VEL
LIN {X 0,Y 343.853,Z 267.275,A -85,B 0,C 180,E1 8446.205,E2 8446.205} C_VEL
LIN {X 0,Y 346.96,Z 272.429,A -85,B 0,C 180,E1 8443.423,E2 8443.423} C_VEL
LIN {X 0,Y 349.811,Z 277.053,A -85,B 0,C 180,E1 8441.329,E2 8441.329} C_VEL
LIN {X 0,Y 353.717,Z 283.366,A -85,B 0,C 180,E1 8438.874,E2 8438.874} C_VEL
LIN {X 0,Y 359.487,Z 293.397,A -85,B 0,C 180,E1 8435.779,E2 8435.779} C_VEL
LIN {X 0,Y 365.717,Z 304.874,A -85,B 0,C 180,E1 8432.922,E2 8432.922} C_VEL
LIN {X 0,Y 366.321,Z 306.441,A -85,B 0,C 180,E1 8432.646,E2 8432.646} C_VEL
LIN {X 0,Y 351.359,Z 514.565,A -85,B 0,C 180,E1 8428.59,E2 8428.59} C_VEL
LIN {X 0,Y 348.337,Z 536.736,A -85,B 0,C 180,E1 8427.994,E2 8427.994} C_VEL
LIN {X 0,Y 344.323,Z 558.075,A -85,B 0,C 180,E1 8427.207,E2 8427.207} C_VEL
LIN {X 0,Y 339.632,Z 577.558,A -85,B 0,C 180,E1 8426.252,E2 8426.252} C_VEL
LIN {X 0,Y 333.504,Z 598.717,A -85,B 0,C 180,E1 8424.929,E2 8424.929} C_VEL
LIN {X 0,Y 326.904,Z 618.22,A -85,B 0,C 180,E1 8423.403,E2 8423.403} C_VEL
LIN {X 0,Y 319.73,Z 636.53,A -85,B 0,C 180,E1 8421.611,E2 8421.611} C_VEL
LIN {X 0,Y 311.863,Z 654.66,A -85,B 0,C 180,E1 8419.448,E2 8419.448} C_VEL
LIN {X 0,Y 304.009,Z 671.153,A -85,B 0,C 180,E1 8417.034,E2 8417.034} C_VEL
LIN {X 0,Y 296.087,Z 686.51,A -85,B 0,C 180,E1 8414.282,E2 8414.282} C_VEL
LIN {X 0,Y 288.413,Z 700.723,A -85,B 0,C 180,E1 8411.198,E2 8411.198} C_VEL
LIN {X 0,Y 281.044,Z 713.684,A -85,B 0,C 180,E1 8407.727,E2 8407.727} C_VEL
LIN {X 0,Y 274.019,Z 725.938,A -85,B 0,C 180,E1 8403.684,E2 8403.684} C_VEL
LIN {X 0,Y 268.239,Z 736.254,A -85,B 0,C 180,E1 8399.473,E2 8399.473} C_VEL
LIN {X 0,Y 263.493,Z 745.039,A -85,B 0,C 180,E1 8394.91,E2 8394.91} C_VEL
LIN {X 0,Y 259.935,Z 752.398,A -85,B 0,C 180,E1 8390.019,E2 8390.019} C_VEL
LIN {X 0,Y 257.773,Z 757.839,A -85,B 0,C 180,E1 8385.293,E2 8385.293} C_VEL
LIN {X 0,Y 256.603,Z 761.619,A -85,B 0,C 180,E1 8380.552,E2 8380.552} C_VEL
LIN {X 0,Y 256.131,Z 764.079,A -85,B 0,C 180,E1 8375.825,E2 8375.825} C_VEL
LIN {X 0,Y 256.018,Z 765.011,A -85,B 0,C 180,E1 8371.566,E2 8371.566} C_VEL
LIN {X 0,Y 256.031,Z 764.917,A -85,B 0,C 180,E1 8367.314,E2 8367.314} C_VEL
LIN {X 0,Y 256.226,Z 763.434,A -85,B 0,C 180,E1 8362.601,E2 8362.601} C_VEL
LIN {X 0,Y 256.88,Z 760.64,A -85,B 0,C 180,E1 8357.867,E2 8357.867} C_VEL
LIN {X 0,Y 258.336,Z 756.266,A -85,B 0,C 180,E1 8353.126,E2 8353.126} C_VEL
LIN {X 0,Y 261.012,Z 750.116,A -85,B 0,C 180,E1 8348.188,E2 8348.188} C_VEL
LIN {X 0,Y 264.851,Z 742.502,A -85,B 0,C 180,E1 8343.547,E2 8343.547} C_VEL
LIN {X 0,Y 270.017,Z 733.032,A -85,B 0,C 180,E1 8339.023,E2 8339.023} C_VEL
LIN {X 0,Y 276.23,Z 722.195,A -85,B 0,C 180,E1 8334.865,E2 8334.865} C_VEL
LIN {X 0,Y 282.866,Z 710.588,A -85,B 0,C 180,E1 8331.271,E2 8331.271} C_VEL
LIN {X 0,Y 290.47,Z 697.015,A -85,B 0,C 180,E1 8327.839,E2 8327.839} C_VEL
LIN {X 0,Y 298.505,Z 682.143,A -85,B 0,C 180,E1 8324.758,E2 8324.758} C_VEL
LIN {X 0,Y 306.421,Z 666.355,A -85,B 0,C 180,E1 8322.114,E2 8322.114} C_VEL
LIN {X 0,Y 314.82,Z 648.25,A -85,B 0,C 180,E1 8319.633,E2 8319.633} C_VEL
LIN {X 0,Y 316.237,Z 645.001,A -85,B 0,C 180,E1 8319.238,E2 8319.238} C_VEL
LIN {X 0,Y 318.22,Z 639.092,A -85,B 0,C 180,E1 8318.401,E2 8318.401} C_VEL
LIN {X 0,Y 320.774,Z 624.318,A -85,B 0,C 180,E1 8315.995,E2 8315.995} C_VEL
LIN {X 0,Y 322.584,Z 617.943,A -85,B 0,C 180,E1 8315.281,E2 8315.281} C_VEL
LIN {X 0,Y 329.134,Z 599.146,A -85,B 0,C 180,E1 8313.816,E2 8313.816} C_VEL
LIN {X 0,Y 335.472,Z 577.966,A -85,B 0,C 180,E1 8312.494,E2 8312.494} C_VEL
LIN {X 0,Y 340.256,Z 558.693,A -85,B 0,C 180,E1 8311.553,E2 8311.553} C_VEL
LIN {X 0,Y 344.509,Z 536.836,A -85,B 0,C 180,E1 8310.75,E2 8310.75} C_VEL
LIN {X 0,Y 347.626,Z 514.669,A -85,B 0,C 180,E1 8310.158,E2 8310.158} C_VEL
LIN {X 0,Y 359.452,Z 355.044,A -85,B 0,C 180,E1 8307.036,E2 8307.036} C_VEL
LIN {X 0,Y 362.799,Z 310.507,A -85,B 0,C 180,E1 8306.165,E2 8306.165} C_VEL
LIN {X 0,Y 356.088,Z 297.975,A -85,B 0,C 180,E1 8302.886,E2 8302.886} C_VEL
LIN {X 0,Y 350.142,Z 287.492,A -85,B 0,C 180,E1 8299.388,E2 8299.388} C_VEL
LIN {X 0,Y 346.156,Z 280.99,A -85,B 0,C 180,E1 8296.53,E2 8296.53} C_VEL
LIN {X 0,Y 343.88,Z 277.211,A -85,B 0,C 180,E1 8294.567,E2 8294.567} C_VEL
LIN {X 0,Y 341.897,Z 273.79,A -85,B 0,C 180,E1 8292.498,E2 8292.498} C_VEL
LIN {X 0,Y 339.311,Z 269.366,A -85,B 0,C 180,E1 8288.814,E2 8288.814} C_VEL
LIN {X 0,Y 337.67,Z 266.138,A -85,B 0,C 180,E1 8282.886,E2 8282.886} C_VEL
LIN {X 0,Y 337.984,Z 266.18,A -85,B 0,C 180,E1 8280,E2 8280} C_VEL
LIN {X 0,Y 340.879,Z 269.707,A -85,B 0,C 180,E1 8274.108,E2 8274.108} C_VEL
LIN {X 0,Y 341.97,Z 271.094,A -85,B 0,C 180,E1 8272.778,E2 8272.778} C_VEL
LIN {X 0,Y 345.641,Z 276.162,A -85,B 0,C 180,E1 8269.247,E2 8269.247} C_VEL
LIN {X 0,Y 349.285,Z 281.476,A -85,B 0,C 180,E1 8266.509,E2 8266.509} C_VEL
LIN {X 0,Y 353.848,Z 288.265,A -85,B 0,C 180,E1 8263.671,E2 8263.671} C_VEL
LIN {X 0,Y 359.676,Z 297.739,A -85,B 0,C 180,E1 8260.598,E2 8260.598} C_VEL
LIN {X 0,Y 364.828,Z 306.602,A -85,B 0,C 180,E1 8258.234,E2 8258.234} C_VEL
LIN {X 0,Y 348.883,Z 506.16,A -85,B 0,C 180,E1 8254.163,E2 8254.163} C_VEL
LIN {X 0,Y 345.966,Z 529.364,A -85,B 0,C 180,E1 8253.573,E2 8253.573} C_VEL
LIN {X 0,Y 341.877,Z 551.399,A -85,B 0,C 180,E1 8252.805,E2 8252.805} C_VEL
LIN {X 0,Y 336.54,Z 574.13,A -85,B 0,C 180,E1 8251.748,E2 8251.748} C_VEL
LIN {X 0,Y 330.518,Z 595.373,A -85,B 0,C 180,E1 8250.484,E2 8250.484} C_VEL
LIN {X 0,Y 323.604,Z 615.939,A -85,B 0,C 180,E1 8248.937,E2 8248.937} C_VEL
LIN {X 0,Y 315.811,Z 636.502,A -85,B 0,C 180,E1 8247.031,E2 8247.031} C_VEL
LIN {X 0,Y 308.177,Z 654.475,A -85,B 0,C 180,E1 8244.988,E2 8244.988} C_VEL
LIN {X 0,Y 299.335,Z 673.573,A -85,B 0,C 180,E1 8242.337,E2 8242.337} C_VEL
LIN {X 0,Y 291.041,Z 690.348,A -85,B 0,C 180,E1 8239.512,E2 8239.512} C_VEL
LIN {X 0,Y 282.602,Z 706.35,A -85,B 0,C 180,E1 8236.198,E2 8236.198} C_VEL
LIN {X 0,Y 274.043,Z 722.237,A -85,B 0,C 180,E1 8232.169,E2 8232.169} C_VEL
LIN {X 0,Y 267.065,Z 735.21,A -85,B 0,C 180,E1 8228.15,E2 8228.15} C_VEL
LIN {X 0,Y 260.966,Z 746.711,A -85,B 0,C 180,E1 8223.747,E2 8223.747} C_VEL
LIN {X 0,Y 255.944,Z 757,A -85,B 0,C 180,E1 8218.948,E2 8218.948} C_VEL
LIN {X 0,Y 252.461,Z 764.959,A -85,B 0,C 180,E1 8214.323,E2 8214.323} C_VEL
LIN {X 0,Y 249.827,Z 772.305,A -85,B 0,C 180,E1 8208.915,E2 8208.915} C_VEL
LIN {X 0,Y 248.587,Z 777.154,A -85,B 0,C 180,E1 8204.202,E2 8204.202} C_VEL
LIN {X 0,Y 248.058,Z 780.743,A -85,B 0,C 180,E1 8199.278,E2 8199.278} C_VEL
LIN {X 0,Y 247.978,Z 782.598,A -85,B 0,C 180,E1 8195.089,E2 8195.089} C_VEL
LIN {X 0,Y 248.003,Z 783.392,A -85,B 0,C 180,E1 8191.025,E2 8191.025} C_VEL
LIN {X 0,Y 247.986,Z 783.101,A -85,B 0,C 180,E1 8186.533,E2 8186.533} C_VEL
LIN {X 0,Y 248.02,Z 781.465,A -85,B 0,C 180,E1 8182.122,E2 8182.122} C_VEL
LIN {X 0,Y 248.318,Z 778.677,A -85,B 0,C 180,E1 8177.678,E2 8177.678} C_VEL
LIN {X 0,Y 249.363,Z 773.9,A -85,B 0,C 180,E1 8172.499,E2 8172.499} C_VEL
LIN {X 0,Y 251.265,Z 768.046,A -85,B 0,C 180,E1 8167.789,E2 8167.789} C_VEL
LIN {X 0,Y 254.774,Z 759.469,A -85,B 0,C 180,E1 8162.414,E2 8162.414} C_VEL
LIN {X 0,Y 259.439,Z 749.784,A -85,B 0,C 180,E1 8157.565,E2 8157.565} C_VEL
LIN {X 0,Y 265.244,Z 738.477,A -85,B 0,C 180,E1 8153.049,E2 8153.049} C_VEL
LIN {X 0,Y 272.465,Z 725.067,A -85,B 0,C 180,E1 8148.66,E2 8148.66} C_VEL
LIN {X 0,Y 279.907,Z 711.357,A -85,B 0,C 180,E1 8144.988,E2 8144.988} C_VEL
LIN {X 0,Y 288.063,Z 695.866,A -85,B 0,C 180,E1 8141.585,E2 8141.585} C_VEL
LIN {X 0,Y 296.584,Z 679.132,A -85,B 0,C 180,E1 8138.546,E2 8138.546} C_VEL
LIN {X 0,Y 304.93,Z 661.507,A -85,B 0,C 180,E1 8135.94,E2 8135.94} C_VEL
LIN {X 0,Y 313.632,Z 641.562,A -85,B 0,C 180,E1 8133.526,E2 8133.526} C_VEL
LIN {X 0,Y 321.188,Z 622.509,A -85,B 0,C 180,E1 8131.638,E2 8131.638} C_VEL
LIN {X 0,Y 328.05,Z 602.709,A -85,B 0,C 180,E1 8130.052,E2 8130.052} C_VEL
LIN {X 0,Y 334.137,Z 582.886,A -85,B 0,C 180,E1 8128.749,E2 8128.749} C_VEL
LIN {X 0,Y 339.476,Z 561.846,A -85,B 0,C 180,E1 8127.662,E2 8127.662} C_VEL
LIN {X 0,Y 344.183,Z 539.18,A -85,B 0,C 180,E1 8126.755,E2 8126.755} C_VEL
LIN {X 0,Y 347.52,Z 517.544,A -85,B 0,C 180,E1 8126.118,E2 8126.118} C_VEL
LIN {X 0,Y 350.465,Z 485.919,A -85,B 0,C 180,E1 8125.418,E2 8125.418} C_VEL
LIN {X 0,Y 364.704,Z 306.434,A -85,B 0,C 180,E1 8121.764,E2 8121.764} C_VEL
LIN {X 0,Y 358.329,Z 295.559,A -85,B 0,C 180,E1 8118.801,E2 8118.801} C_VEL
LIN {X 0,Y 352.63,Z 286.577,A -85,B 0,C 180,E1 8115.711,E2 8115.711} C_VEL
LIN {X 0,Y 348.003,Z 279.549,A -85,B 0,C 180,E1 8112.697,E2 8112.697} C_VEL
LIN {X 0,Y 344.426,Z 274.563,A -85,B 0,C 180,E1 8109.862,E2 8109.862} C_VEL
LIN {X 0,Y 341.1,Z 269.95,A -85,B 0,C 180,E1 8106.395,E2 8106.395} C_VEL
LIN {X 0,Y 337.788,Z 265.836,A -85,B 0,C 180,E1 8100,E2 8100} C_VEL
LIN {X 0,Y 337.457,Z 265.71,A -85,B 0,C 180,E1 8097.283,E2 8097.283} C_VEL
LIN {X 0,Y 338.606,Z 268.627,A -85,B 0,C 180,E1 8092.022,E2 8092.022} C_VEL
LIN {X 0,Y 339.597,Z 270.003,A -85,B 0,C 180,E1 8090.253,E2 8090.253} C_VEL
LIN {X 0,Y 342.559,Z 274.988,A -85,B 0,C 180,E1 8086.496,E2 8086.496} C_VEL
LIN {X 0,Y 345.582,Z 280.16,A -85,B 0,C 180,E1 8083.701,E2 8083.701} C_VEL
LIN {X 0,Y 348.254,Z 284.626,A -85,B 0,C 180,E1 8081.676,E2 8081.676} C_VEL
LIN {X 0,Y 351.934,Z 290.774,A -85,B 0,C 180,E1 8079.285,E2 8079.285} C_VEL
LIN {X 0,Y 357.501,Z 300.693,A -85,B 0,C 180,E1 8076.206,E2 8076.206} C_VEL
LIN {X 0,Y 362.7,Z 310.709,A -85,B 0,C 180,E1 8073.713,E2 8073.713} C_VEL
LIN {X 0,Y 347.52,Z 514.548,A -85,B 0,C 180,E1 8069.745,E2 8069.745} C_VEL
LIN {X 0,Y 344.424,Z 536.655,A -85,B 0,C 180,E1 8069.155,E2 8069.155} C_VEL
LIN {X 0,Y 340.256,Z 558.222,A -85,B 0,C 180,E1 8068.367,E2 8068.367} C_VEL
LIN {X 0,Y 335.344,Z 578.042,A -85,B 0,C 180,E1 8067.4,E2 8067.4} C_VEL
LIN {X 0,Y 328.974,Z 599.32,A -85,B 0,C 180,E1 8066.069,E2 8066.069} C_VEL
LIN {X 0,Y 322.186,Z 618.748,A -85,B 0,C 180,E1 8064.548,E2 8064.548} C_VEL
LIN {X 0,Y 314.696,Z 637.231,A -85,B 0,C 180,E1 8062.734,E2 8062.734} C_VEL
LIN {X 0,Y 306.089,Z 656.271,A -85,B 0,C 180,E1 8060.433,E2 8060.433} C_VEL
LIN {X 0,Y 297.735,Z 673.157,A -85,B 0,C 180,E1 8057.914,E2 8057.914} C_VEL
LIN {X 0,Y 289.441,Z 688.462,A -85,B 0,C 180,E1 8055.084,E2 8055.084} C_VEL
LIN {X 0,Y 280.963,Z 703.311,A -85,B 0,C 180,E1 8051.717,E2 8051.717} C_VEL
LIN {X 0,Y 273.443,Z 716.059,A -85,B 0,C 180,E1 8048.166,E2 8048.166} C_VEL
LIN {X 0,Y 266.57,Z 727.366,A -85,B 0,C 180,E1 8044.236,E2 8044.236} C_VEL
LIN {X 0,Y 260.322,Z 737.887,A -85,B 0,C 180,E1 8039.7,E2 8039.7} C_VEL
LIN {X 0,Y 255.491,Z 746.514,A -85,B 0,C 180,E1 8035.002,E2 8035.002} C_VEL
LIN {X 0,Y 251.872,Z 753.567,A -85,B 0,C 180,E1 8029.961,E2 8029.961} C_VEL
LIN {X 0,Y 249.548,Z 759.122,A -85,B 0,C 180,E1 8024.62,E2 8024.62} C_VEL
LIN {X 0,Y 248.487,Z 762.668,A -85,B 0,C 180,E1 8019.729,E2 8019.729} C_VEL
LIN {X 0,Y 248.093,Z 764.688,A -85,B 0,C 180,E1 8014.855,E2 8014.855} C_VEL
LIN {X 0,Y 248.02,Z 765.409,A -85,B 0,C 180,E1 8010.462,E2 8010.462} C_VEL
LIN {X 0,Y 248.072,Z 764.909,A -85,B 0,C 180,E1 8005.84,E2 8005.84} C_VEL
LIN {X 0,Y 248.335,Z 763.301,A -85,B 0,C 180,E1 8001.433,E2 8001.433} C_VEL
LIN {X 0,Y 249.257,Z 759.997,A -85,B 0,C 180,E1 7996.31,E2 7996.31} C_VEL
LIN {X 0,Y 251.217,Z 755.115,A -85,B 0,C 180,E1 7991.193,E2 7991.193} C_VEL
LIN {X 0,Y 254.47,Z 748.392,A -85,B 0,C 180,E1 7986.128,E2 7986.128} C_VEL
LIN {X 0,Y 259.317,Z 739.656,A -85,B 0,C 180,E1 7981.075,E2 7981.075} C_VEL
LIN {X 0,Y 265.172,Z 729.829,A -85,B 0,C 180,E1 7976.599,E2 7976.599} C_VEL
LIN {X 0,Y 271.798,Z 718.796,A -85,B 0,C 180,E1 7972.618,E2 7972.618} C_VEL
LIN {X 0,Y 279.504,Z 705.892,A -85,B 0,C 180,E1 7968.837,E2 7968.837} C_VEL
LIN {X 0,Y 287.833,Z 691.566,A -85,B 0,C 180,E1 7965.438,E2 7965.438} C_VEL
LIN {X 0,Y 295.972,Z 676.562,A -85,B 0,C 180,E1 7962.572,E2 7962.572} C_VEL
LIN {X 0,Y 304.784,Z 659.169,A -85,B 0,C 180,E1 7959.859,E2 7959.859} C_VEL
LIN {X 0,Y 313.024,Z 641.441,A -85,B 0,C 180,E1 7957.614,E2 7957.614} C_VEL
LIN {X 0,Y 320.744,Z 622.628,A -85,B 0,C 180,E1 7955.705,E2 7955.705} C_VEL
LIN {X 0,Y 322.584,Z 617.943,A -85,B 0,C 180,E1 7955.281,E2 7955.281} C_VEL
LIN {X 0,Y 324.38,Z 611.451,A -85,B 0,C 180,E1 7954.593,E2 7954.593} C_VEL
LIN {X 0,Y 326.75,Z 595.409,A -85,B 0,C 180,E1 7952.496,E2 7952.496} C_VEL
LIN {X 0,Y 328.322,Z 588.624,A -85,B 0,C 180,E1 7951.91,E2 7951.91} C_VEL
LIN {X 0,Y 334.124,Z 568.06,A -85,B 0,C 180,E1 7950.778,E2 7950.778} C_VEL
LIN {X 0,Y 338.871,Z 546.87,A -85,B 0,C 180,E1 7949.896,E2 7949.896} C_VEL
LIN {X 0,Y 342.735,Z 523.976,A -85,B 0,C 180,E1 7949.205,E2 7949.205} C_VEL
LIN {X 0,Y 345.182,Z 500.961,A -85,B 0,C 180,E1 7948.689,E2 7948.689} C_VEL
LIN {X 0,Y 359.299,Z 315.137,A -85,B 0,C 180,E1 7945.09,E2 7945.09} C_VEL
LIN {X 0,Y 353.448,Z 304.02,A -85,B 0,C 180,E1 7942.057,E2 7942.057} C_VEL
LIN {X 0,Y 348.141,Z 294.371,A -85,B 0,C 180,E1 7938.764,E2 7938.764} C_VEL
LIN {X 0,Y 344.384,Z 288.046,A -85,B 0,C 180,E1 7935.924,E2 7935.924} C_VEL
LIN {X 0,Y 342.222,Z 284.362,A -85,B 0,C 180,E1 7933.948,E2 7933.948} C_VEL
LIN {X 0,Y 340.638,Z 281.504,A -85,B 0,C 180,E1 7932.201,E2 7932.201} C_VEL
LIN {X 0,Y 338.254,Z 277.252,A -85,B 0,C 180,E1 7928.671,E2 7928.671} C_VEL
LIN {X 0,Y 336.699,Z 274.04,A -85,B 0,C 180,E1 7922.724,E2 7922.724} C_VEL
LIN {X 0,Y 337.008,Z 274.129,A -85,B 0,C 180,E1 7920,E2 7920} C_VEL
LIN {X 0,Y 340.154,Z 277.964,A -85,B 0,C 180,E1 7913.756,E2 7913.756} C_VEL
LIN {X 0,Y 344.151,Z 283.69,A -85,B 0,C 180,E1 7909.623,E2 7909.623} C_VEL
LIN {X 0,Y 347.799,Z 289.181,A -85,B 0,C 180,E1 7906.789,E2 7906.789} C_VEL
LIN {X 0,Y 352.201,Z 295.972,A -85,B 0,C 180,E1 7903.974,E2 7903.974} C_VEL
LIN {X 0,Y 357.693,Z 305.123,A -85,B 0,C 180,E1 7900.995,E2 7900.995} C_VEL
LIN {X 0,Y 361.202,Z 311.452,A -85,B 0,C 180,E1 7899.298,E2 7899.298} C_VEL
LIN {X 0,Y 345.079,Z 507.25,A -85,B 0,C 180,E1 7895.315,E2 7895.315} C_VEL
LIN {X 0,Y 341.95,Z 530.805,A -85,B 0,C 180,E1 7894.708,E2 7894.708} C_VEL
LIN {X 0,Y 337.791,Z 552.49,A -85,B 0,C 180,E1 7893.952,E2 7893.952} C_VEL
LIN {X 0,Y 332.392,Z 574.667,A -85,B 0,C 180,E1 7892.919,E2 7892.919} C_VEL
LIN {X 0,Y 326.093,Z 596.22,A -85,B 0,C 180,E1 7891.638,E2 7891.638} C_VEL
LIN {X 0,Y 319.037,Z 616.469,A -85,B 0,C 180,E1 7890.113,E2 7890.113} C_VEL
LIN {X 0,Y 310.745,Z 637.526,A -85,B 0,C 180,E1 7888.149,E2 7888.149} C_VEL
LIN {X 0,Y 302.61,Z 656.004,A -85,B 0,C 180,E1 7886.028,E2 7886.028} C_VEL
LIN {X 0,Y 294.03,Z 673.741,A -85,B 0,C 180,E1 7883.533,E2 7883.533} C_VEL
LIN {X 0,Y 285.482,Z 690.358,A -85,B 0,C 180,E1 7880.714,E2 7880.714} C_VEL
LIN {X 0,Y 276.864,Z 705.99,A -85,B 0,C 180,E1 7877.451,E2 7877.451} C_VEL
LIN {X 0,Y 268.294,Z 721.175,A -85,B 0,C 180,E1 7873.585,E2 7873.585} C_VEL
LIN {X 0,Y 260.861,Z 734.218,A -85,B 0,C 180,E1 7869.512,E2 7869.512} C_VEL
LIN {X 0,Y 254.325,Z 745.852,A -85,B 0,C 180,E1 7865.028,E2 7865.028} C_VEL
LIN {X 0,Y 248.901,Z 756.221,A -85,B 0,C 180,E1 7860.14,E2 7860.14} C_VEL
LIN {X 0,Y 244.9,Z 764.648,A -85,B 0,C 180,E1 7855.125,E2 7855.125} C_VEL
LIN {X 0,Y 242.034,Z 772.002,A -85,B 0,C 180,E1 7849.549,E2 7849.549} C_VEL
LIN {X 0,Y 240.668,Z 776.854,A -85,B 0,C 180,E1 7844.68,E2 7844.68} C_VEL
LIN {X 0,Y 240.075,Z 780.448,A -85,B 0,C 180,E1 7839.589,E2 7839.589} C_VEL
LIN {X 0,Y 239.981,Z 782.306,A -85,B 0,C 180,E1 7835.259,E2 7835.259} C_VEL
LIN {X 0,Y 240.009,Z 783.097,A -85,B 0,C 180,E1 7831.101,E2 7831.101} C_VEL
LIN {X 0,Y 239.988,Z 782.809,A -85,B 0,C 180,E1 7826.417,E2 7826.417} C_VEL
LIN {X 0,Y 240.03,Z 781.17,A -85,B 0,C 180,E1 7821.858,E2 7821.858} C_VEL
LIN {X 0,Y 240.365,Z 778.379,A -85,B 0,C 180,E1 7817.264,E2 7817.264} C_VEL
LIN {X 0,Y 241.526,Z 773.595,A -85,B 0,C 180,E1 7811.912,E2 7811.912} C_VEL
LIN {X 0,Y 243.596,Z 767.738,A -85,B 0,C 180,E1 7807.05,E2 7807.05} C_VEL
LIN {X 0,Y 247.2,Z 759.576,A -85,B 0,C 180,E1 7801.756,E2 7801.756} C_VEL
LIN {X 0,Y 251.815,Z 750.507,A -85,B 0,C 180,E1 7797.047,E2 7797.047} C_VEL
LIN {X 0,Y 258.081,Z 739.023,A -85,B 0,C 180,E1 7792.258,E2 7792.258} C_VEL
LIN {X 0,Y 265.412,Z 726.169,A -85,B 0,C 180,E1 7787.891,E2 7787.891} C_VEL
LIN {X 0,Y 273.116,Z 712.593,A -85,B 0,C 180,E1 7784.15,E2 7784.15} C_VEL
LIN {X 0,Y 282.062,Z 696.441,A -85,B 0,C 180,E1 7780.506,E2 7780.506} C_VEL
LIN {X 0,Y 290.904,Z 679.854,A -85,B 0,C 180,E1 7777.445,E2 7777.445} C_VEL
LIN {X 0,Y 299.651,Z 662.069,A -85,B 0,C 180,E1 7774.79,E2 7774.79} C_VEL
LIN {X 0,Y 308.505,Z 642.576,A -85,B 0,C 180,E1 7772.408,E2 7772.408} C_VEL
LIN {X 0,Y 315.943,Z 624.467,A -85,B 0,C 180,E1 7770.597,E2 7770.597} C_VEL
LIN {X 0,Y 323.331,Z 604.129,A -85,B 0,C 180,E1 7768.942,E2 7768.942} C_VEL
LIN {X 0,Y 329.57,Z 584.512,A -85,B 0,C 180,E1 7767.643,E2 7767.643} C_VEL
LIN {X 0,Y 335.241,Z 563.121,A -85,B 0,C 180,E1 7766.527,E2 7766.527} C_VEL
LIN {X 0,Y 340.046,Z 541.061,A -85,B 0,C 180,E1 7765.632,E2 7765.632} C_VEL
LIN {X 0,Y 343.621,Z 518.746,A -85,B 0,C 180,E1 7764.972,E2 7764.972} C_VEL
LIN {X 0,Y 346.653,Z 487.925,A -85,B 0,C 180,E1 7764.285,E2 7764.285} C_VEL
LIN {X 0,Y 361.08,Z 311.128,A -85,B 0,C 180,E1 7760.695,E2 7760.695} C_VEL
LIN {X 0,Y 355.118,Z 300.887,A -85,B 0,C 180,E1 7757.745,E2 7757.745} C_VEL
LIN {X 0,Y 350.179,Z 292.914,A -85,B 0,C 180,E1 7754.89,E2 7754.89} C_VEL
LIN {X 0,Y 345.887,Z 286.388,A -85,B 0,C 180,E1 7751.928,E2 7751.928} C_VEL
LIN {X 0,Y 343.059,Z 282.249,A -85,B 0,C 180,E1 7749.563,E2 7749.563} C_VEL
LIN {X 0,Y 339.903,Z 277.751,A -85,B 0,C 180,E1 7746.156,E2 7746.156} C_VEL
LIN {X 0,Y 336.81,Z 273.788,A -85,B 0,C 180,E1 7740,E2 7740} C_VEL
LIN {X 0,Y 336.482,Z 273.663,A -85,B 0,C 180,E1 7737.275,E2 7737.275} C_VEL
LIN {X 0,Y 337.901,Z 276.936,A -85,B 0,C 180,E1 7731.492,E2 7731.492} C_VEL
LIN {X 0,Y 338.565,Z 278.068,A -85,B 0,C 180,E1 7730.309,E2 7730.309} C_VEL
LIN {X 0,Y 341.268,Z 282.699,A -85,B 0,C 180,E1 7726.789,E2 7726.789} C_VEL
LIN {X 0,Y 344.214,Z 287.889,A -85,B 0,C 180,E1 7723.981,E2 7723.981} C_VEL
LIN {X 0,Y 347.391,Z 293.328,A -85,B 0,C 180,E1 7721.542,E2 7721.542} C_VEL
LIN {X 0,Y 352.146,Z 301.684,A -85,B 0,C 180,E1 7718.514,E2 7718.514} C_VEL
LIN {X 0,Y 358.03,Z 312.82,A -85,B 0,C 180,E1 7715.367,E2 7715.367} C_VEL
LIN {X 0,Y 359.185,Z 315.254,A -85,B 0,C 180,E1 7714.796,E2 7714.796} C_VEL
LIN {X 0,Y 343.827,Z 514.492,A -85,B 0,C 180,E1 7710.926,E2 7710.926} C_VEL
LIN {X 0,Y 340.623,Z 536.781,A -85,B 0,C 180,E1 7710.336,E2 7710.336} C_VEL
LIN {X 0,Y 336.329,Z 558.362,A -85,B 0,C 180,E1 7709.554,E2 7709.554} C_VEL
LIN {X 0,Y 331.421,Z 577.677,A -85,B 0,C 180,E1 7708.622,E2 7708.622} C_VEL
LIN {X 0,Y 324.917,Z 598.927,A -85,B 0,C 180,E1 7707.31,E2 7707.31} C_VEL
LIN {X 0,Y 317.927,Z 618.424,A -85,B 0,C 180,E1 7705.801,E2 7705.801} C_VEL
LIN {X 0,Y 310.21,Z 636.957,A -85,B 0,C 180,E1 7703.998,E2 7703.998} C_VEL
LIN {X 0,Y 301.608,Z 655.482,A -85,B 0,C 180,E1 7701.781,E2 7701.781} C_VEL
LIN {X 0,Y 293.22,Z 671.895,A -85,B 0,C 180,E1 7699.36,E2 7699.36} C_VEL
LIN {X 0,Y 284.781,Z 687.015,A -85,B 0,C 180,E1 7696.615,E2 7696.615} C_VEL
LIN {X 0,Y 276.34,Z 701.398,A -85,B 0,C 180,E1 7693.428,E2 7693.428} C_VEL
LIN {X 0,Y 268.23,Z 714.45,A -85,B 0,C 180,E1 7689.835,E2 7689.835} C_VEL
LIN {X 0,Y 260.544,Z 726.576,A -85,B 0,C 180,E1 7685.683,E2 7685.683} C_VEL
LIN {X 0,Y 254.094,Z 736.873,A -85,B 0,C 180,E1 7681.292,E2 7681.292} C_VEL
LIN {X 0,Y 248.735,Z 745.655,A -85,B 0,C 180,E1 7676.499,E2 7676.499} C_VEL
LIN {X 0,Y 244.613,Z 753.088,A -85,B 0,C 180,E1 7671.258,E2 7671.258} C_VEL
LIN {X 0,Y 242.042,Z 758.639,A -85,B 0,C 180,E1 7666.067,E2 7666.067} C_VEL
LIN {X 0,Y 240.694,Z 762.359,A -85,B 0,C 180,E1 7661.016,E2 7661.016} C_VEL
LIN {X 0,Y 240.153,Z 764.726,A -85,B 0,C 180,E1 7655.974,E2 7655.974} C_VEL
LIN {X 0,Y 240.029,Z 765.614,A -85,B 0,C 180,E1 7651.432,E2 7651.432} C_VEL
LIN {X 0,Y 240.05,Z 765.478,A -85,B 0,C 180,E1 7646.896,E2 7646.896} C_VEL
LIN {X 0,Y 240.286,Z 763.987,A -85,B 0,C 180,E1 7642.034,E2 7642.034} C_VEL
LIN {X 0,Y 241.072,Z 761.228,A -85,B 0,C 180,E1 7637.058,E2 7637.058} C_VEL
LIN {X 0,Y 242.798,Z 756.861,A -85,B 0,C 180,E1 7632.01,E2 7632.01} C_VEL
LIN {X 0,Y 245.915,Z 750.711,A -85,B 0,C 180,E1 7626.764,E2 7626.764} C_VEL
LIN {X 0,Y 250.285,Z 743.109,A -85,B 0,C 180,E1 7621.876,E2 7621.876} C_VEL
LIN {X 0,Y 256.098,Z 733.654,A -85,B 0,C 180,E1 7617.135,E2 7617.135} C_VEL
LIN {X 0,Y 263,Z 722.838,A -85,B 0,C 180,E1 7612.81,E2 7612.81} C_VEL
LIN {X 0,Y 270.301,Z 711.24,A -85,B 0,C 180,E1 7609.102,E2 7609.102} C_VEL
LIN {X 0,Y 278.631,Z 697.634,A -85,B 0,C 180,E1 7605.57,E2 7605.57} C_VEL
LIN {X 0,Y 287.292,Z 682.868,A -85,B 0,C 180,E1 7602.456,E2 7602.456} C_VEL
LIN {X 0,Y 295.886,Z 666.955,A -85,B 0,C 180,E1 7599.759,E2 7599.759} C_VEL
LIN {X 0,Y 305.074,Z 648.449,A -85,B 0,C 180,E1 7597.213,E2 7597.213} C_VEL
LIN {X 0,Y 313.225,Z 630.312,A -85,B 0,C 180,E1 7595.198,E2 7595.198} C_VEL
LIN {X 0,Y 320.781,Z 610.994,A -85,B 0,C 180,E1 7593.484,E2 7593.484} C_VEL
LIN {X 0,Y 327.805,Z 590.313,A -85,B 0,C 180,E1 7592.014,E2 7592.014} C_VEL
LIN {X 0,Y 328.322,Z 588.624,A -85,B 0,C 180,E1 7591.91,E2 7591.91} C_VEL
LIN {X 0,Y 329.994,Z 581.723,A -85,B 0,C 180,E1 7591.355,E2 7591.355} C_VEL
LIN {X 0,Y 331.675,Z 564.579,A -85,B 0,C 180,E1 7589.56,E2 7589.56} C_VEL
LIN {X 0,Y 332.933,Z 557.459,A -85,B 0,C 180,E1 7589.085,E2 7589.085} C_VEL
LIN {X 0,Y 337.295,Z 535.764,A -85,B 0,C 180,E1 7588.322,E2 7588.322} C_VEL
LIN {X 0,Y 340.561,Z 512.908,A -85,B 0,C 180,E1 7587.735,E2 7587.735} C_VEL
LIN {X 0,Y 355.926,Z 319.841,A -85,B 0,C 180,E1 7583.998,E2 7583.998} C_VEL
LIN {X 0,Y 350.303,Z 308.855,A -85,B 0,C 180,E1 7580.859,E2 7580.859} C_VEL
LIN {X 0,Y 345.896,Z 300.855,A -85,B 0,C 180,E1 7577.93,E2 7577.93} C_VEL
LIN {X 0,Y 342.836,Z 295.434,A -85,B 0,C 180,E1 7575.477,E2 7575.477} C_VEL
LIN {X 0,Y 339.709,Z 289.632,A -85,B 0,C 180,E1 7572.275,E2 7572.275} C_VEL
LIN {X 0,Y 337.107,Z 285.041,A -85,B 0,C 180,E1 7568.357,E2 7568.357} C_VEL
LIN {X 0,Y 335.723,Z 281.993,A -85,B 0,C 180,E1 7562.732,E2 7562.732} C_VEL
LIN {X 0,Y 336.032,Z 282.081,A -85,B 0,C 180,E1 7560,E2 7560} C_VEL
LIN {X 0,Y 339.17,Z 285.96,A -85,B 0,C 180,E1 7553.738,E2 7553.738} C_VEL
LIN {X 0,Y 342.856,Z 291.531,A -85,B 0,C 180,E1 7549.838,E2 7549.838} C_VEL
LIN {X 0,Y 346.325,Z 296.885,A -85,B 0,C 180,E1 7547.071,E2 7547.071} C_VEL
LIN {X 0,Y 350.503,Z 303.557,A -85,B 0,C 180,E1 7544.319,E2 7544.319} C_VEL
LIN {X 0,Y 355.728,Z 312.502,A -85,B 0,C 180,E1 7541.397,E2 7541.397} C_VEL
LIN {X 0,Y 357.704,Z 316.31,A -85,B 0,C 180,E1 7540.383,E2 7540.383} C_VEL
LIN {X 0,Y 341.415,Z 508.375,A -85,B 0,C 180,E1 7536.49,E2 7536.49} C_VEL
LIN {X 0,Y 337.895,Z 533.243,A -85,B 0,C 180,E1 7535.837,E2 7535.837} C_VEL
LIN {X 0,Y 333.539,Z 555.073,A -85,B 0,C 180,E1 7535.065,E2 7535.065} C_VEL
LIN {X 0,Y 328.024,Z 576.506,A -85,B 0,C 180,E1 7534.049,E2 7534.049} C_VEL
LIN {X 0,Y 321.564,Z 597.668,A -85,B 0,C 180,E1 7532.779,E2 7532.779} C_VEL
LIN {X 0,Y 314.225,Z 618.028,A -85,B 0,C 180,E1 7531.236,E2 7531.236} C_VEL
LIN {X 0,Y 305.801,Z 638.553,A -85,B 0,C 180,E1 7529.304,E2 7529.304} C_VEL
LIN {X 0,Y 297.115,Z 657.599,A -85,B 0,C 180,E1 7527.098,E2 7527.098} C_VEL
LIN {X 0,Y 288.268,Z 675.045,A -85,B 0,C 180,E1 7524.595,E2 7524.595} C_VEL
LIN {X 0,Y 279.158,Z 691.9,A -85,B 0,C 180,E1 7521.662,E2 7521.662} C_VEL
LIN {X 0,Y 270.767,Z 706.503,A -85,B 0,C 180,E1 7518.555,E2 7518.555} C_VEL
LIN {X 0,Y 261.828,Z 721.559,A -85,B 0,C 180,E1 7514.638,E2 7514.638} C_VEL
LIN {X 0,Y 254.058,Z 734.541,A -85,B 0,C 180,E1 7510.492,E2 7510.492} C_VEL
LIN {X 0,Y 247.184,Z 746.067,A -85,B 0,C 180,E1 7505.91,E2 7505.91} C_VEL
LIN {X 0,Y 241.457,Z 756.332,A -85,B 0,C 180,E1 7500.895,E2 7500.895} C_VEL
LIN {X 0,Y 237.383,Z 764.339,A -85,B 0,C 180,E1 7495.979,E2 7495.979} C_VEL
LIN {X 0,Y 234.272,Z 771.699,A -85,B 0,C 180,E1 7490.224,E2 7490.224} C_VEL
LIN {X 0,Y 232.763,Z 776.554,A -85,B 0,C 180,E1 7485.19,E2 7485.19} C_VEL
LIN {X 0,Y 232.094,Z 780.154,A -85,B 0,C 180,E1 7479.922,E2 7479.922} C_VEL
LIN {X 0,Y 231.984,Z 782.014,A -85,B 0,C 180,E1 7475.441,E2 7475.441} C_VEL
LIN {X 0,Y 232.014,Z 782.804,A -85,B 0,C 180,E1 7471.167,E2 7471.167} C_VEL
LIN {X 0,Y 231.994,Z 782.571,A -85,B 0,C 180,E1 7466.541,E2 7466.541} C_VEL
LIN {X 0,Y 232.035,Z 780.875,A -85,B 0,C 180,E1 7461.576,E2 7461.576} C_VEL
LIN {X 0,Y 232.42,Z 778.081,A -85,B 0,C 180,E1 7456.821,E2 7456.821} C_VEL
LIN {X 0,Y 233.712,Z 773.291,A -85,B 0,C 180,E1 7451.285,E2 7451.285} C_VEL
LIN {X 0,Y 235.987,Z 767.386,A -85,B 0,C 180,E1 7446.23,E2 7446.23} C_VEL
LIN {X 0,Y 240.089,Z 758.836,A -85,B 0,C 180,E1 7440.567,E2 7440.567} C_VEL
LIN {X 0,Y 245.392,Z 749.225,A -85,B 0,C 180,E1 7435.504,E2 7435.504} C_VEL
LIN {X 0,Y 251.843,Z 738.098,A -85,B 0,C 180,E1 7430.858,E2 7430.858} C_VEL
LIN {X 0,Y 259.854,Z 724.776,A -85,B 0,C 180,E1 7426.334,E2 7426.334} C_VEL
LIN {X 0,Y 267.818,Z 711.448,A -85,B 0,C 180,E1 7422.655,E2 7422.655} C_VEL
LIN {X 0,Y 276.965,Z 695.591,A -85,B 0,C 180,E1 7419.092,E2 7419.092} C_VEL
LIN {X 0,Y 286.205,Z 678.885,A -85,B 0,C 180,E1 7416.029,E2 7416.029} C_VEL
LIN {X 0,Y 294.912,Z 661.805,A -85,B 0,C 180,E1 7413.488,E2 7413.488} C_VEL
LIN {X 0,Y 304.297,Z 641.756,A -85,B 0,C 180,E1 7411.055,E2 7411.055} C_VEL
LIN {X 0,Y 312.171,Z 623.127,A -85,B 0,C 180,E1 7409.218,E2 7409.218} C_VEL
LIN {X 0,Y 319.667,Z 602.835,A -85,B 0,C 180,E1 7407.602,E2 7407.602} C_VEL
LIN {X 0,Y 326.216,Z 582.643,A -85,B 0,C 180,E1 7406.299,E2 7406.299} C_VEL
LIN {X 0,Y 331.861,Z 561.494,A -85,B 0,C 180,E1 7405.231,E2 7405.231} C_VEL
LIN {X 0,Y 336.799,Z 538.715,A -85,B 0,C 180,E1 7404.348,E2 7404.348} C_VEL
LIN {X 0,Y 340.271,Z 517.096,A -85,B 0,C 180,E1 7403.727,E2 7403.727} C_VEL
LIN {X 0,Y 343.446,Z 484.305,A -85,B 0,C 180,E1 7403.012,E2 7403.012} C_VEL
LIN {X 0,Y 357.573,Z 315.957,A -85,B 0,C 180,E1 7399.606,E2 7399.606} C_VEL
LIN {X 0,Y 352.174,Z 306.421,A -85,B 0,C 180,E1 7396.748,E2 7396.748} C_VEL
LIN {X 0,Y 347.212,Z 298.318,A -85,B 0,C 180,E1 7393.658,E2 7393.658} C_VEL
LIN {X 0,Y 343.843,Z 293.187,A -85,B 0,C 180,E1 7391.15,E2 7391.15} C_VEL
LIN {X 0,Y 341.614,Z 289.83,A -85,B 0,C 180,E1 7389.178,E2 7389.178} C_VEL
LIN {X 0,Y 338.718,Z 285.563,A -85,B 0,C 180,E1 7385.93,E2 7385.93} C_VEL
LIN {X 0,Y 335.791,Z 281.684,A -85,B 0,C 180,E1 7379.829,E2 7379.829} C_VEL
LIN {X 0,Y 335.506,Z 281.616,A -85,B 0,C 180,E1 7377.267,E2 7377.267} C_VEL
LIN {X 0,Y 337.179,Z 285.172,A -85,B 0,C 180,E1 7371.043,E2 7371.043} C_VEL
LIN {X 0,Y 339.987,Z 290.41,A -85,B 0,C 180,E1 7367.085,E2 7367.085} C_VEL
LIN {X 0,Y 342.851,Z 295.616,A -85,B 0,C 180,E1 7364.263,E2 7364.263} C_VEL
LIN {X 0,Y 346.539,Z 302.009,A -85,B 0,C 180,E1 7361.408,E2 7361.408} C_VEL
LIN {X 0,Y 351.965,Z 312.199,A -85,B 0,C 180,E1 7357.976,E2 7357.976} C_VEL
LIN {X 0,Y 355.788,Z 319.958,A -85,B 0,C 180,E1 7355.897,E2 7355.897} C_VEL
LIN {X 0,Y 340.287,Z 514.4,A -85,B 0,C 180,E1 7352.132,E2 7352.132} C_VEL
LIN {X 0,Y 336.999,Z 536.729,A -85,B 0,C 180,E1 7351.547,E2 7351.547} C_VEL
LIN {X 0,Y 332.552,Z 558.502,A -85,B 0,C 180,E1 7350.768,E2 7350.768} C_VEL
LIN {X 0,Y 327.343,Z 578.432,A -85,B 0,C 180,E1 7349.813,E2 7349.813} C_VEL
LIN {X 0,Y 320.669,Z 599.525,A -85,B 0,C 180,E1 7348.513,E2 7348.513} C_VEL
LIN {X 0,Y 313.489,Z 618.945,A -85,B 0,C 180,E1 7347.014,E2 7347.014} C_VEL
LIN {X 0,Y 305.548,Z 637.42,A -85,B 0,C 180,E1 7345.219,E2 7345.219} C_VEL
LIN {X 0,Y 296.368,Z 656.489,A -85,B 0,C 180,E1 7342.926,E2 7342.926} C_VEL
LIN {X 0,Y 287.405,Z 673.4,A -85,B 0,C 180,E1 7340.404,E2 7340.404} C_VEL
LIN {X 0,Y 278.372,Z 688.859,A -85,B 0,C 180,E1 7337.525,E2 7337.525} C_VEL
LIN {X 0,Y 269,Z 703.986,A -85,B 0,C 180,E1 7334.031,E2 7334.031} C_VEL
LIN {X 0,Y 260.773,Z 716.719,A -85,B 0,C 180,E1 7330.388,E2 7330.388} C_VEL
LIN {X 0,Y 253.193,Z 728.002,A -85,B 0,C 180,E1 7326.323,E2 7326.323} C_VEL
LIN {X 0,Y 245.921,Z 738.947,A -85,B 0,C 180,E1 7321.359,E2 7321.359} C_VEL
LIN {X 0,Y 240.528,Z 747.49,A -85,B 0,C 180,E1 7316.409,E2 7316.409} C_VEL
LIN {X 0,Y 236.446,Z 754.46,A -85,B 0,C 180,E1 7311.065,E2 7311.065} C_VEL
LIN {X 0,Y 233.874,Z 759.716,A -85,B 0,C 180,E1 7305.624,E2 7305.624} C_VEL
LIN {X 0,Y 232.605,Z 763.258,A -85,B 0,C 180,E1 7300.401,E2 7300.401} C_VEL
LIN {X 0,Y 232.12,Z 765.271,A -85,B 0,C 180,E1 7295.19,E2 7295.19} C_VEL
LIN {X 0,Y 232.03,Z 765.991,A -85,B 0,C 180,E1 7290.494,E2 7290.494} C_VEL
LIN {X 0,Y 232.092,Z 765.492,A -85,B 0,C 180,E1 7285.553,E2 7285.553} C_VEL
LIN {X 0,Y 232.424,Z 763.886,A -85,B 0,C 180,E1 7280.842,E2 7280.842} C_VEL
LIN {X 0,Y 233.526,Z 760.588,A -85,B 0,C 180,E1 7275.368,E2 7275.368} C_VEL
LIN {X 0,Y 235.697,Z 755.95,A -85,B 0,C 180,E1 7270.162,E2 7270.162} C_VEL
LIN {X 0,Y 239.388,Z 749.333,A -85,B 0,C 180,E1 7264.785,E2 7264.785} C_VEL
LIN {X 0,Y 244.69,Z 740.908,A -85,B 0,C 180,E1 7259.557,E2 7259.557} C_VEL
LIN {X 0,Y 251.294,Z 730.98,A -85,B 0,C 180,E1 7254.766,E2 7254.766} C_VEL
LIN {X 0,Y 258.953,Z 719.462,A -85,B 0,C 180,E1 7250.426,E2 7250.426} C_VEL
LIN {X 0,Y 267.9,Z 705.808,A -85,B 0,C 180,E1 7246.335,E2 7246.335} C_VEL
LIN {X 0,Y 276.461,Z 692.262,A -85,B 0,C 180,E1 7243.068,E2 7243.068} C_VEL
LIN {X 0,Y 285.246,Z 677.269,A -85,B 0,C 180,E1 7240.163,E2 7240.163} C_VEL
LIN {X 0,Y 294.678,Z 659.973,A -85,B 0,C 180,E1 7237.444,E2 7237.444} C_VEL
LIN {X 0,Y 303.455,Z 642.302,A -85,B 0,C 180,E1 7235.203,E2 7235.203} C_VEL
LIN {X 0,Y 311.308,Z 624.407,A -85,B 0,C 180,E1 7233.38,E2 7233.38} C_VEL
LIN {X 0,Y 318.782,Z 605.292,A -85,B 0,C 180,E1 7231.792,E2 7231.792} C_VEL
LIN {X 0,Y 325.057,Z 586.482,A -85,B 0,C 180,E1 7230.544,E2 7230.544} C_VEL
LIN {X 0,Y 331.009,Z 565.292,A -85,B 0,C 180,E1 7229.431,E2 7229.431} C_VEL
LIN {X 0,Y 332.933,Z 557.459,A -85,B 0,C 180,E1 7229.085,E2 7229.085} C_VEL
LIN {X 0,Y 334.168,Z 550.238,A -85,B 0,C 180,E1 7228.637,E2 7228.637} C_VEL
LIN {X 0,Y 334.928,Z 532.17,A -85,B 0,C 180,E1 7227.126,E2 7227.126} C_VEL
LIN {X 0,Y 335.633,Z 524.721,A -85,B 0,C 180,E1 7226.785,E2 7226.785} C_VEL
LIN {X 0,Y 338.246,Z 502.025,A -85,B 0,C 180,E1 7226.277,E2 7226.277} C_VEL
LIN {X 0,Y 352.626,Z 324.598,A -85,B 0,C 180,E1 7222.859,E2 7222.859} C_VEL
LIN {X 0,Y 348.03,Z 315.337,A -85,B 0,C 180,E1 7220.123,E2 7220.123} C_VEL
LIN {X 0,Y 344.153,Z 308.052,A -85,B 0,C 180,E1 7217.412,E2 7217.412} C_VEL
LIN {X 0,Y 340.539,Z 301.241,A -85,B 0,C 180,E1 7214.279,E2 7214.279} C_VEL
LIN {X 0,Y 338.148,Z 296.93,A -85,B 0,C 180,E1 7211.6,E2 7211.6} C_VEL
LIN {X 0,Y 336.056,Z 292.926,A -85,B 0,C 180,E1 7208.211,E2 7208.211} C_VEL
LIN {X 0,Y 334.75,Z 289.896,A -85,B 0,C 180,E1 7202.568,E2 7202.568} C_VEL
LIN {X 0,Y 335.055,Z 290.035,A -85,B 0,C 180,E1 7200,E2 7200} C_VEL
LIN {X 0,Y 337.986,Z 293.77,A -85,B 0,C 180,E1 7193.972,E2 7193.972} C_VEL
LIN {X 0,Y 341.567,Z 299.369,A -85,B 0,C 180,E1 7190.055,E2 7190.055} C_VEL
LIN {X 0,Y 344.972,Z 304.767,A -85,B 0,C 180,E1 7187.275,E2 7187.275} C_VEL
LIN {X 0,Y 349.198,Z 311.813,A -85,B 0,C 180,E1 7184.429,E2 7184.429} C_VEL
LIN {X 0,Y 354.356,Z 320.893,A -85,B 0,C 180,E1 7181.499,E2 7181.499} C_VEL
LIN {X 0,Y 338.041,Z 508.147,A -85,B 0,C 180,E1 7177.721,E2 7177.721} C_VEL
LIN {X 0,Y 334.548,Z 532.537,A -85,B 0,C 180,E1 7177.094,E2 7177.094} C_VEL
LIN {X 0,Y 330.037,Z 554.709,A -85,B 0,C 180,E1 7176.325,E2 7176.325} C_VEL
LIN {X 0,Y 324.262,Z 576.685,A -85,B 0,C 180,E1 7175.298,E2 7175.298} C_VEL
LIN {X 0,Y 317.569,Z 597.986,A -85,B 0,C 180,E1 7174.03,E2 7174.03} C_VEL
LIN {X 0,Y 309.996,Z 618.397,A -85,B 0,C 180,E1 7172.493,E2 7172.493} C_VEL
LIN {X 0,Y 301.421,Z 638.619,A -85,B 0,C 180,E1 7170.598,E2 7170.598} C_VEL
LIN {X 0,Y 292.365,Z 657.819,A -85,B 0,C 180,E1 7168.379,E2 7168.379} C_VEL
LIN {X 0,Y 283.054,Z 675.521,A -85,B 0,C 180,E1 7165.83,E2 7165.83} C_VEL
LIN {X 0,Y 272.913,Z 693.434,A -85,B 0,C 180,E1 7162.654,E2 7162.654} C_VEL
LIN {X 0,Y 263.74,Z 708.757,A -85,B 0,C 180,E1 7159.303,E2 7159.303} C_VEL
LIN {X 0,Y 254.999,Z 722.669,A -85,B 0,C 180,E1 7155.529,E2 7155.529} C_VEL
LIN {X 0,Y 246.933,Z 735.45,A -85,B 0,C 180,E1 7151.299,E2 7151.299} C_VEL
LIN {X 0,Y 239.782,Z 746.815,A -85,B 0,C 180,E1 7146.603,E2 7146.603} C_VEL
LIN {X 0,Y 233.562,Z 757.291,A -85,B 0,C 180,E1 7141.197,E2 7141.197} C_VEL
LIN {X 0,Y 229.047,Z 765.87,A -85,B 0,C 180,E1 7135.604,E2 7135.604} C_VEL
LIN {X 0,Y 226.211,Z 772.203,A -85,B 0,C 180,E1 7130.167,E2 7130.167} C_VEL
LIN {X 0,Y 224.654,Z 777.113,A -85,B 0,C 180,E1 7124.695,E2 7124.695} C_VEL
LIN {X 0,Y 224.071,Z 780.225,A -85,B 0,C 180,E1 7119.503,E2 7119.503} C_VEL
LIN {X 0,Y 223.987,Z 781.868,A -85,B 0,C 180,E1 7115.122,E2 7115.122} C_VEL
LIN {X 0,Y 224.017,Z 782.578,A -85,B 0,C 180,E1 7110.511,E2 7110.511} C_VEL
LIN {X 0,Y 223.989,Z 782.08,A -85,B 0,C 180,E1 7105.648,E2 7105.648} C_VEL
LIN {X 0,Y 224.049,Z 780.459,A -85,B 0,C 180,E1 7101.014,E2 7101.014} C_VEL
LIN {X 0,Y 224.521,Z 777.612,A -85,B 0,C 180,E1 7096.086,E2 7096.086} C_VEL
LIN {X 0,Y 226.01,Z 772.717,A -85,B 0,C 180,E1 7090.354,E2 7090.354} C_VEL
LIN {X 0,Y 228.551,Z 766.803,A -85,B 0,C 180,E1 7085.168,E2 7085.168} C_VEL
LIN {X 0,Y 232.845,Z 758.521,A -85,B 0,C 180,E1 7079.556,E2 7079.556} C_VEL
LIN {X 0,Y 238.521,Z 748.903,A -85,B 0,C 180,E1 7074.362,E2 7074.362} C_VEL
LIN {X 0,Y 245.378,Z 737.77,A -85,B 0,C 180,E1 7069.619,E2 7069.619} C_VEL
LIN {X 0,Y 253.643,Z 724.758,A -85,B 0,C 180,E1 7065.122,E2 7065.122} C_VEL
LIN {X 0,Y 262.202,Z 711.099,A -85,B 0,C 180,E1 7061.305,E2 7061.305} C_VEL
LIN {X 0,Y 271.771,Z 695.22,A -85,B 0,C 180,E1 7057.724,E2 7057.724} C_VEL
LIN {X 0,Y 281.085,Z 679.049,A -85,B 0,C 180,E1 7054.747,E2 7054.747} C_VEL
LIN {X 0,Y 290.243,Z 661.708,A -85,B 0,C 180,E1 7052.165,E2 7052.165} C_VEL
LIN {X 0,Y 299.958,Z 641.618,A -85,B 0,C 180,E1 7049.738,E2 7049.738} C_VEL
LIN {X 0,Y 308.267,Z 622.533,A -85,B 0,C 180,E1 7047.873,E2 7047.873} C_VEL
LIN {X 0,Y 316.028,Z 601.984,A -85,B 0,C 180,E1 7046.265,E2 7046.265} C_VEL
LIN {X 0,Y 323.035,Z 580.578,A -85,B 0,C 180,E1 7044.924,E2 7044.924} C_VEL
LIN {X 0,Y 328.653,Z 559.862,A -85,B 0,C 180,E1 7043.91,E2 7043.91} C_VEL
LIN {X 0,Y 333.674,Z 536.637,A -85,B 0,C 180,E1 7043.047,E2 7043.047} C_VEL
LIN {X 0,Y 337.286,Z 514.026,A -85,B 0,C 180,E1 7042.42,E2 7042.42} C_VEL
LIN {X 0,Y 342.892,Z 451.52,A -85,B 0,C 180,E1 7041.124,E2 7041.124} C_VEL
LIN {X 0,Y 354.161,Z 320.675,A -85,B 0,C 180,E1 7038.475,E2 7038.475} C_VEL
LIN {X 0,Y 348.734,Z 311.127,A -85,B 0,C 180,E1 7035.379,E2 7035.379} C_VEL
LIN {X 0,Y 344.708,Z 304.45,A -85,B 0,C 180,E1 7032.65,E2 7032.65} C_VEL
LIN {X 0,Y 340.893,Z 298.247,A -85,B 0,C 180,E1 7029.453,E2 7029.453} C_VEL
LIN {X 0,Y 337.601,Z 293.434,A -85,B 0,C 180,E1 7025.779,E2 7025.779} C_VEL
LIN {X 0,Y 334.775,Z 289.581,A -85,B 0,C 180,E1 7019.657,E2 7019.657} C_VEL
LIN {X 0,Y 334.532,Z 289.622,A -85,B 0,C 180,E1 7017.087,E2 7017.087} C_VEL
LIN {X 0,Y 336.192,Z 293.346,A -85,B 0,C 180,E1 7011.017,E2 7011.017} C_VEL
LIN {X 0,Y 338.792,Z 298.272,A -85,B 0,C 180,E1 7007.298,E2 7007.298} C_VEL
LIN {X 0,Y 341.501,Z 303.341,A -85,B 0,C 180,E1 7004.548,E2 7004.548} C_VEL
LIN {X 0,Y 345.21,Z 310.053,A -85,B 0,C 180,E1 7001.596,E2 7001.596} C_VEL
LIN {X 0,Y 350.079,Z 319.513,A -85,B 0,C 180,E1 6998.425,E2 6998.425} C_VEL
LIN {X 0,Y 352.502,Z 324.807,A -85,B 0,C 180,E1 6997.017,E2 6997.017} C_VEL
LIN {X 0,Y 336.898,Z 514.329,A -85,B 0,C 180,E1 6993.363,E2 6993.363} C_VEL
LIN {X 0,Y 333.528,Z 536.677,A -85,B 0,C 180,E1 6992.785,E2 6992.785} C_VEL
LIN {X 0,Y 328.927,Z 558.638,A -85,B 0,C 180,E1 6992.009,E2 6992.009} C_VEL
LIN {X 0,Y 323.769,Z 577.913,A -85,B 0,C 180,E1 6991.101,E2 6991.101} C_VEL
LIN {X 0,Y 316.921,Z 599.128,A -85,B 0,C 180,E1 6989.817,E2 6989.817} C_VEL
LIN {X 0,Y 309.541,Z 618.619,A -85,B 0,C 180,E1 6988.333,E2 6988.333} C_VEL
LIN {X 0,Y 301.361,Z 637.156,A -85,B 0,C 180,E1 6986.554,E2 6986.554} C_VEL
LIN {X 0,Y 292.209,Z 655.698,A -85,B 0,C 180,E1 6984.354,E2 6984.354} C_VEL
LIN {X 0,Y 283.209,Z 672.173,A -85,B 0,C 180,E1 6981.931,E2 6981.931} C_VEL
LIN {X 0,Y 273.862,Z 687.729,A -85,B 0,C 180,E1 6979.089,E2 6979.089} C_VEL
LIN {X 0,Y 264.723,Z 702.068,A -85,B 0,C 180,E1 6975.857,E2 6975.857} C_VEL
LIN {X 0,Y 255.956,Z 715.007,A -85,B 0,C 180,E1 6972.212,E2 6972.212} C_VEL
LIN {X 0,Y 247.419,Z 727.21,A -85,B 0,C 180,E1 6967.897,E2 6967.897} C_VEL
LIN {X 0,Y 240.235,Z 737.488,A -85,B 0,C 180,E1 6963.324,E2 6963.324} C_VEL
LIN {X 0,Y 234.193,Z 746.268,A -85,B 0,C 180,E1 6958.287,E2 6958.287} C_VEL
LIN {X 0,Y 229.515,Z 753.604,A -85,B 0,C 180,E1 6952.812,E2 6952.812} C_VEL
LIN {X 0,Y 226.46,Z 759.232,A -85,B 0,C 180,E1 6947.206,E2 6947.206} C_VEL
LIN {X 0,Y 224.848,Z 762.95,A -85,B 0,C 180,E1 6941.803,E2 6941.803} C_VEL
LIN {X 0,Y 224.192,Z 765.31,A -85,B 0,C 180,E1 6936.401,E2 6936.401} C_VEL
LIN {X 0,Y 224.041,Z 766.174,A -85,B 0,C 180,E1 6931.79,E2 6931.79} C_VEL
LIN {X 0,Y 224.054,Z 766.101,A -85,B 0,C 180,E1 6927.186,E2 6927.186} C_VEL
LIN {X 0,Y 224.321,Z 764.712,A -85,B 0,C 180,E1 6921.8,E2 6921.8} C_VEL
LIN {X 0,Y 225.174,Z 762.116,A -85,B 0,C 180,E1 6916.65,E2 6916.65} C_VEL
LIN {X 0,Y 227.229,Z 757.697,A -85,B 0,C 180,E1 6910.998,E2 6910.998} C_VEL
LIN {X 0,Y 230.766,Z 751.664,A -85,B 0,C 180,E1 6905.422,E2 6905.422} C_VEL
LIN {X 0,Y 235.679,Z 744.105,A -85,B 0,C 180,E1 6900.241,E2 6900.241} C_VEL
LIN {X 0,Y 242.154,Z 734.752,A -85,B 0,C 180,E1 6895.253,E2 6895.253} C_VEL
LIN {X 0,Y 249.736,Z 724.093,A -85,B 0,C 180,E1 6890.761,E2 6890.761} C_VEL
LIN {X 0,Y 258.158,Z 711.887,A -85,B 0,C 180,E1 6886.724,E2 6886.724} C_VEL
LIN {X 0,Y 267.714,Z 697.56,A -85,B 0,C 180,E1 6882.946,E2 6882.946} C_VEL
LIN {X 0,Y 277.158,Z 682.623,A -85,B 0,C 180,E1 6879.791,E2 6879.791} C_VEL
LIN {X 0,Y 286.407,Z 666.626,A -85,B 0,C 180,E1 6877.091,E2 6877.091} C_VEL
LIN {X 0,Y 295.914,Z 648.64,A -85,B 0,C 180,E1 6874.641,E2 6874.641} C_VEL
LIN {X 0,Y 304.578,Z 630.488,A -85,B 0,C 180,E1 6872.647,E2 6872.647} C_VEL
LIN {X 0,Y 312.514,Z 611.322,A -85,B 0,C 180,E1 6870.972,E2 6870.972} C_VEL
LIN {X 0,Y 320.129,Z 590.056,A -85,B 0,C 180,E1 6869.492,E2 6869.492} C_VEL
LIN {X 0,Y 326.483,Z 568.904,A -85,B 0,C 180,E1 6868.339,E2 6868.339} C_VEL
LIN {X 0,Y 331.511,Z 547.643,A -85,B 0,C 180,E1 6867.469,E2 6867.469} C_VEL
LIN {X 0,Y 335.633,Z 524.721,A -85,B 0,C 180,E1 6866.785,E2 6866.785} C_VEL
LIN {X 0,Y 336.334,Z 517.223,A -85,B 0,C 180,E1 6866.459,E2 6866.459} C_VEL
LIN {X 0,Y 335.71,Z 497.617,A -85,B 0,C 180,E1 6865.06,E2 6865.06} C_VEL
LIN {X 0,Y 335.935,Z 491.115,A -85,B 0,C 180,E1 6864.815,E2 6864.815} C_VEL
LIN {X 0,Y 349.477,Z 329.321,A -85,B 0,C 180,E1 6861.707,E2 6861.707} C_VEL
LIN {X 0,Y 344.993,Z 320.16,A -85,B 0,C 180,E1 6858.81,E2 6858.81} C_VEL
LIN {X 0,Y 342.035,Z 314.489,A -85,B 0,C 180,E1 6856.56,E2 6856.56} C_VEL
LIN {X 0,Y 338.979,Z 308.548,A -85,B 0,C 180,E1 6853.736,E2 6853.736} C_VEL
LIN {X 0,Y 336.917,Z 304.642,A -85,B 0,C 180,E1 6851.296,E2 6851.296} C_VEL
LIN {X 0,Y 335.008,Z 300.812,A -85,B 0,C 180,E1 6848.064,E2 6848.064} C_VEL
LIN {X 0,Y 333.779,Z 297.798,A -85,B 0,C 180,E1 6842.404,E2 6842.404} C_VEL
LIN {X 0,Y 334.114,Z 298.069,A -85,B 0,C 180,E1 6839.829,E2 6839.829} C_VEL
LIN {X 0,Y 336.866,Z 301.678,A -85,B 0,C 180,E1 6834.123,E2 6834.123} C_VEL
LIN {X 0,Y 340.195,Z 307.051,A -85,B 0,C 180,E1 6830.356,E2 6830.356} C_VEL
LIN {X 0,Y 343.516,Z 312.472,A -85,B 0,C 180,E1 6827.562,E2 6827.562} C_VEL
LIN {X 0,Y 347.77,Z 319.821,A -85,B 0,C 180,E1 6824.62,E2 6824.62} C_VEL
LIN {X 0,Y 351.106,Z 326.062,A -85,B 0,C 180,E1 6822.617,E2 6822.617} C_VEL
LIN {X 0,Y 334.542,Z 510.567,A -85,B 0,C 180,E1 6818.918,E2 6818.918} C_VEL
LIN {X 0,Y 330.928,Z 534.184,A -85,B 0,C 180,E1 6818.301,E2 6818.301} C_VEL
LIN {X 0,Y 326.187,Z 556.587,A -85,B 0,C 180,E1 6817.52,E2 6817.52} C_VEL
LIN {X 0,Y 320.445,Z 577.597,A -85,B 0,C 180,E1 6816.537,E2 6816.537} C_VEL
LIN {X 0,Y 312.906,Z 600.543,A -85,B 0,C 180,E1 6815.157,E2 6815.157} C_VEL
LIN {X 0,Y 304.842,Z 621.499,A -85,B 0,C 180,E1 6813.559,E2 6813.559} C_VEL
LIN {X 0,Y 296.305,Z 640.61,A -85,B 0,C 180,E1 6811.727,E2 6811.727} C_VEL
LIN {X 0,Y 286.762,Z 659.891,A -85,B 0,C 180,E1 6809.451,E2 6809.451} C_VEL
LIN {X 0,Y 277.684,Z 676.523,A -85,B 0,C 180,E1 6807.028,E2 6807.028} C_VEL
LIN {X 0,Y 267.34,Z 694.021,A -85,B 0,C 180,E1 6803.884,E2 6803.884} C_VEL
LIN {X 0,Y 257.813,Z 709.272,A -85,B 0,C 180,E1 6800.504,E2 6800.504} C_VEL
LIN {X 0,Y 248.707,Z 723.052,A -85,B 0,C 180,E1 6796.689,E2 6796.689} C_VEL
LIN {X 0,Y 239.672,Z 736.581,A -85,B 0,C 180,E1 6792.049,E2 6792.049} C_VEL
LIN {X 0,Y 232.086,Z 748.098,A -85,B 0,C 180,E1 6787.094,E2 6787.094} C_VEL
LIN {X 0,Y 225.925,Z 757.825,A -85,B 0,C 180,E1 6781.778,E2 6781.778} C_VEL
LIN {X 0,Y 221.208,Z 766.208,A -85,B 0,C 180,E1 6776.004,E2 6776.004} C_VEL
LIN {X 0,Y 218.254,Z 772.437,A -85,B 0,C 180,E1 6770.375,E2 6770.375} C_VEL
LIN {X 0,Y 216.598,Z 777.329,A -85,B 0,C 180,E1 6764.434,E2 6764.434} C_VEL
LIN {X 0,Y 216.063,Z 780.175,A -85,B 0,C 180,E1 6759.321,E2 6759.321} C_VEL
LIN {X 0,Y 215.992,Z 781.794,A -85,B 0,C 180,E1 6754.513,E2 6754.513} C_VEL
LIN {X 0,Y 216.022,Z 782.285,A -85,B 0,C 180,E1 6749.47,E2 6749.47} C_VEL
LIN {X 0,Y 215.991,Z 781.569,A -85,B 0,C 180,E1 6744.688,E2 6744.688} C_VEL
LIN {X 0,Y 216.09,Z 779.92,A -85,B 0,C 180,E1 6740.143,E2 6740.143} C_VEL
LIN {X 0,Y 216.808,Z 776.592,A -85,B 0,C 180,E1 6734.486,E2 6734.486} C_VEL
LIN {X 0,Y 218.591,Z 771.608,A -85,B 0,C 180,E1 6728.817,E2 6728.817} C_VEL
LIN {X 0,Y 221.93,Z 764.794,A -85,B 0,C 180,E1 6722.934,E2 6722.934} C_VEL
LIN {X 0,Y 226.701,Z 756.514,A -85,B 0,C 180,E1 6717.448,E2 6717.448} C_VEL
LIN {X 0,Y 233.43,Z 745.908,A -85,B 0,C 180,E1 6711.918,E2 6711.918} C_VEL
LIN {X 0,Y 241.101,Z 734.461,A -85,B 0,C 180,E1 6707.149,E2 6707.149} C_VEL
LIN {X 0,Y 249.657,Z 721.525,A -85,B 0,C 180,E1 6702.872,E2 6702.872} C_VEL
LIN {X 0,Y 259.429,Z 706.556,A -85,B 0,C 180,E1 6698.877,E2 6698.877} C_VEL
LIN {X 0,Y 268.803,Z 691.529,A -85,B 0,C 180,E1 6695.637,E2 6695.637} C_VEL
LIN {X 0,Y 278.637,Z 674.627,A -85,B 0,C 180,E1 6692.691,E2 6692.691} C_VEL
LIN {X 0,Y 288.084,Z 657.214,A -85,B 0,C 180,E1 6690.21,E2 6690.21} C_VEL
LIN {X 0,Y 297.335,Z 638.152,A -85,B 0,C 180,E1 6688.031,E2 6688.031} C_VEL
LIN {X 0,Y 306.629,Z 616.678,A -85,B 0,C 180,E1 6686.061,E2 6686.061} C_VEL
LIN {X 0,Y 314.389,Z 596.17,A -85,B 0,C 180,E1 6684.557,E2 6684.557} C_VEL
LIN {X 0,Y 321.19,Z 574.62,A -85,B 0,C 180,E1 6683.321,E2 6683.321} C_VEL
LIN {X 0,Y 327.382,Z 550.662,A -85,B 0,C 180,E1 6682.261,E2 6682.261} C_VEL
LIN {X 0,Y 331.959,Z 527.905,A -85,B 0,C 180,E1 6681.52,E2 6681.52} C_VEL
LIN {X 0,Y 335.033,Z 504.714,A -85,B 0,C 180,E1 6680.964,E2 6680.964} C_VEL
LIN {X 0,Y 350.98,Z 325.816,A -85,B 0,C 180,E1 6677.387,E2 6677.387} C_VEL
LIN {X 0,Y 346.213,Z 317.114,A -85,B 0,C 180,E1 6674.466,E2 6674.466} C_VEL
LIN {X 0,Y 341.82,Z 309.701,A -85,B 0,C 180,E1 6671.216,E2 6671.216} C_VEL
LIN {X 0,Y 338.941,Z 305.199,A -85,B 0,C 180,E1 6668.567,E2 6668.567} C_VEL
LIN {X 0,Y 336.364,Z 301.174,A -85,B 0,C 180,E1 6665.458,E2 6665.458} C_VEL
